KUKA KRL program: MyProgram_057().src

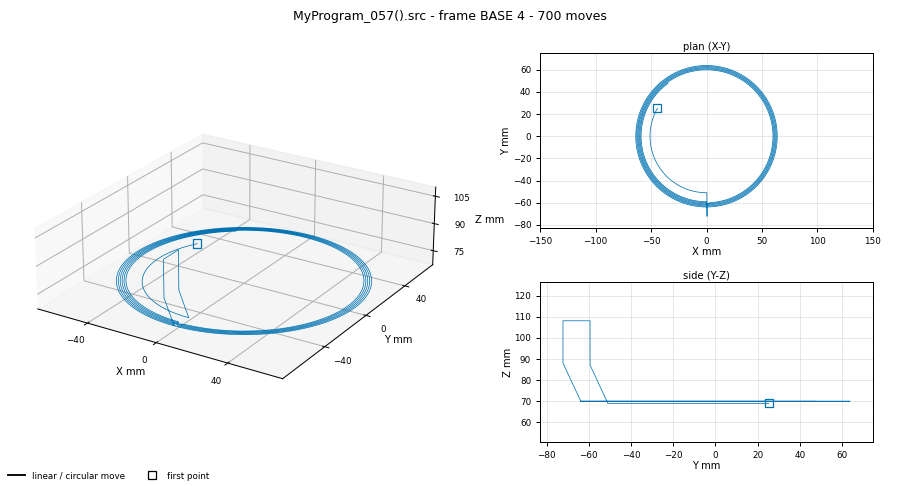
[picture p0: tool path of MyProgram_057().src in frame BASE 4, 700 of 700 moves have a stored position in this frame; points joined in program order, loops and branches not executed]
&ACCESS RVP
&REL 1
&PARAM TEMPLATE = C:\KRC\Roboter\Template\vorgabe
&PARAM EDITMASK = *
DEF MyProgram_057()
; ---- Setting reference (Base) ----
$BASE = BASE_DATA[4]

; --------------------------
; ---- Setting tool (TCP) ----
$TOOL = TOOL_DATA[3]
; --------------------------

$VEL.CP = VEL_APROX_PRINT
Startdeposition()
$VEL.CP = VEL_PRINT
LIN {X -44.2675,Y 25.2093,Z 69,A 144.3707,B 24.8543,C -2.785,E1 24.86,E2 299.1753} C_DIS
LIN {X -45.377,Y 23.1519,Z 69,A 147.0437,B 24.855,C -2.7781,E1 24.8565,E2 296.5045} C_DIS
LIN {X -46.4551,Y 20.9046,Z 69,A 149.9054,B 24.8558,C -2.7707,E1 24.8531,E2 293.6449} C_DIS
LIN {X -47.4216,Y 18.6083,Z 69,A 152.7265,B 24.8566,C -2.7626,E1 24.8502,E2 290.8275} C_DIS
LIN {X -48.2606,Y 16.3092,Z 69,A 155.5004,B 24.8575,C -2.7546,E1 24.8476,E2 288.057} C_DIS
LIN {X -49.0262,Y 13.8387,Z 69,A 158.4298,B 24.8584,C -2.7459,E1 24.8453,E2 285.1313} C_DIS
LIN {X -49.6447,Y 11.4229,Z 69,A 161.2158,B 24.8593,C -2.7369,E1 24.8435,E2 282.3505} C_DIS
LIN {X -50.1315,Y 9.0506,Z 69,A 163.9981,B 24.8601,C -2.7293,E1 24.842,E2 279.5701} C_DIS
LIN {X -50.5144,Y 6.5863,Z 69,A 166.8631,B 24.8609,C -2.7213,E1 24.8409,E2 276.707} C_DIS
LIN {X -50.7819,Y 4.0351,Z 69,A 169.7378,B 24.8619,C -2.7121,E1 24.8401,E2 273.8372} C_DIS
LIN {X -50.9193,Y 1.5178,Z 69,A 172.5271,B 24.8628,C -2.7025,E1 24.8398,E2 271.0541} C_DIS
LIN {X -50.9339,Y -0.9051,Z 69,A 175.3708,B 24.8635,C -2.6956,E1 24.8398,E2 268.2097} C_DIS
LIN {X -50.8236,Y -3.4697,Z 69,A 178.24,B 24.8645,C -2.6863,E1 24.8403,E2 265.3454} C_DIS
LIN {X -50.6012,Y -5.8824,Z 69,A -178.9757,B 24.8652,C -2.6787,E1 24.8411,E2 262.5626} C_DIS
LIN {X -50.2495,Y -8.3704,Z 69,A -176.13,B 24.8661,C -2.6703,E1 24.8423,E2 259.7201} C_DIS
LIN {X -49.7641,Y -10.891,Z 69,A -173.3005,B 24.8671,C -2.6607,E1 24.8439,E2 256.8968} C_DIS
LIN {X -49.1711,Y -13.3146,Z 69,A -170.4355,B 24.8678,C -2.6532,E1 24.8459,E2 254.0332} C_DIS
LIN {X -48.4775,Y -15.6528,Z 69,A -167.6344,B 24.8685,C -2.646,E1 24.8482,E2 251.2332} C_DIS
LIN {X -47.6271,Y -18.076,Z 69,A -164.8739,B 24.8696,C -2.6358,E1 24.8509,E2 248.4814} C_DIS
LIN {X -46.7092,Y -20.3305,Z 69,A -162.0822,B 24.8702,C -2.6289,E1 24.8539,E2 245.6908} C_DIS
LIN {X -45.6565,Y -22.5956,Z 69,A -159.1445,B 24.8708,C -2.6231,E1 24.8574,E2 242.751} C_DIS
LIN {X -44.4616,Y -24.8646,Z 69,A -156.2811,B 24.8716,C -2.6151,E1 24.8612,E2 239.8916} C_DIS
LIN {X -43.1923,Y -27.0093,Z 69,A -153.5018,B 24.8723,C -2.6075,E1 24.8653,E2 237.1162} C_DIS
LIN {X -41.8616,Y -29.0291,Z 69,A -150.6713,B 24.8728,C -2.6024,E1 24.8697,E2 234.2837} C_DIS
LIN {X -40.3456,Y -31.1016,Z 69,A -147.7568,B 24.8735,C -2.5959,E1 24.8746,E2 231.3707} C_DIS
LIN {X -38.6707,Y -33.1615,Z 69,A -144.8211,B 24.8742,C -2.5884,E1 24.8798,E2 228.4396} C_DIS
LIN {X -37.0149,Y -35,Z 69,A -142.0063,B 24.8748,C -2.5829,E1 24.8852,E2 225.6255} C_DIS
LIN {X -35.2304,Y -36.7958,Z 69,A -139.1593,B 24.8753,C -2.577,E1 24.8908,E2 222.7805} C_DIS
LIN {X -33.3921,Y -38.4716,Z 69,A -136.3039,B 24.8758,C -2.5726,E1 24.8968,E2 219.9244} C_DIS
LIN {X -31.3436,Y -40.1591,Z 69,A -133.3517,B 24.8763,C -2.5667,E1 24.9032,E2 216.9753} C_DIS
LIN {X -29.3388,Y -41.6462,Z 69,A -130.5429,B 24.8768,C -2.562,E1 24.9096,E2 214.1678} C_DIS
LIN {X -27.2507,Y -43.0415,Z 69,A -127.7018,B 24.8772,C -2.558,E1 24.9162,E2 211.3271} C_DIS
LIN {X -25.1158,Y -44.3212,Z 69,A -124.8909,B 24.8775,C -2.5543,E1 24.923,E2 208.5166} C_DIS
LIN {X -22.9218,Y -45.4946,Z 69,A -122.0757,B 24.8778,C -2.5511,E1 24.93,E2 205.7013} C_DIS
LIN {X -20.6449,Y -46.5721,Z 69,A -119.2428,B 24.8781,C -2.5479,E1 24.9372,E2 202.869} C_DIS
LIN {X -18.3398,Y -47.5271,Z 69,A -116.4302,B 24.8784,C -2.5453,E1 24.9445,E2 200.0564} C_DIS
LIN {X -15.9911,Y -48.3679,Z 69,A -113.6192,B 24.8786,C -2.5432,E1 24.9519,E2 197.2451} C_DIS
LIN {X -13.5856,Y -49.0979,Z 69,A -110.7884,B 24.8788,C -2.5413,E1 24.9595,E2 194.4141} C_DIS
LIN {X -11.1685,Y -49.7035,Z 69,A -107.9816,B 24.8788,C -2.54,E1 24.9671,E2 191.6066} C_DIS
LIN {X -8.7255,Y -50.19,Z 69,A -105.1777,B 24.879,C -2.5391,E1 24.9748,E2 188.802} C_DIS
LIN {X -6.264,Y -50.5561,Z 69,A -102.3662,B 24.879,C -2.5387,E1 24.9826,E2 185.9891} C_DIS
LIN {X -3.751,Y -50.8046,Z 69,A -99.5364,B 24.879,C -2.5384,E1 24.9905,E2 183.1587} C_DIS
LIN {X -1.2642,Y -50.9271,Z 69,A -96.7368,B 24.879,C -2.5387,E1 24.9983,E2 180.3579} C_DIS
LIN {X 0.3002,Y -50.939,Z 69,A -95.324,B 24.8796,C -2.5329,E1 25.0022,E2 178.9589} C_DIS
Enddeposition()
LIN {X 0.3252,Y -53.0519,Z 73.5315,A -95.3128,B 24.88,C -2.5282,E1 25.0022,E2 178.9589} C_DIS
LIN {X 0.4003,Y -59.3907,Z 87.1262,A -95.2837,B 24.8812,C -2.516,E1 25.0022,E2 178.9589} C_DIS
LIN {X 0.4003,Y -59.3907,Z 108.1262,A -95.6377,B 24.8666,C -2.6649,E1 25.0022,E2 178.9589} C_DIS
LIN {X 0.5021,Y -72.2249,Z 108.1262,A -95.1125,B 24.8869,C -2.4543,E1 25.0022,E2 178.9342} C_DIS
LIN {X 0.5021,Y -72.2249,Z 88.1262,A -94.7756,B 24.8997,C -2.3125,E1 25.0022,E2 178.9342} C_DIS
LIN {X 0.4243,Y -65.8861,Z 74.5315,A -94.8025,B 24.8987,C -2.3239,E1 25.0022,E2 178.9342} C_DIS
LIN {X 0.3983,Y -63.7731,Z 70,A -94.813,B 24.8983,C -2.3283,E1 25.0022,E2 178.9342} C_DIS
Startdeposition()
$VEL.CP = VEL_PRINT
LIN {X 3.1294,Y -63.7012,Z 70,A -92.0208,B 24.8975,C -2.3368,E1 25.0101,E2 176.1225} C_DIS
LIN {X 6.2513,Y -63.4709,Z 70,A -89.2116,B 24.8975,C -2.3382,E1 25.0179,E2 173.3116} C_DIS
LIN {X 9.3582,Y -63.0877,Z 70,A -86.4031,B 24.8973,C -2.3399,E1 25.0257,E2 170.5014} C_DIS
LIN {X 12.4425,Y -62.5525,Z 70,A -83.5957,B 24.8971,C -2.3421,E1 25.0334,E2 167.6921} C_DIS
LIN {X 15.4968,Y -61.8667,Z 70,A -80.7893,B 24.8969,C -2.3446,E1 25.0411,E2 164.8836} C_DIS
LIN {X 18.5138,Y -61.0318,Z 70,A -77.9838,B 24.8966,C -2.3475,E1 25.0486,E2 162.0759} C_DIS
LIN {X 21.4862,Y -60.0498,Z 70,A -75.1792,B 24.8963,C -2.3509,E1 25.056,E2 159.269} C_DIS
LIN {X 24.4068,Y -58.9232,Z 70,A -72.3755,B 24.896,C -2.3545,E1 25.0633,E2 156.4629} C_DIS
LIN {X 27.2686,Y -57.6546,Z 70,A -69.5725,B 24.8956,C -2.3586,E1 25.0704,E2 153.6573} C_DIS
LIN {X 30.0647,Y -56.2472,Z 70,A -66.7706,B 24.8952,C -2.363,E1 25.0773,E2 150.8527} C_DIS
LIN {X 32.7885,Y -54.7042,Z 70,A -63.9694,B 24.8948,C -2.3678,E1 25.0841,E2 148.0488} C_DIS
LIN {X 35.4332,Y -53.0295,Z 70,A -61.1691,B 24.8943,C -2.3729,E1 25.0907,E2 145.2456} C_DIS
LIN {X 37.9925,Y -51.227,Z 70,A -58.3694,B 24.8939,C -2.3783,E1 25.097,E2 142.443} C_DIS
LIN {X 40.4603,Y -49.3011,Z 70,A -55.5704,B 24.8933,C -2.384,E1 25.1031,E2 139.6409} C_DIS
LIN {X 42.8307,Y -47.2564,Z 70,A -52.7723,B 24.8928,C -2.39,E1 25.109,E2 136.8397} C_DIS
LIN {X 45.0979,Y -45.0979,Z 70,A -49.9747,B 24.8922,C -2.3963,E1 25.1146,E2 134.0389} C_DIS
LIN {X 47.2564,Y -42.8307,Z 70,A -47.1669,B 24.8916,C -2.4032,E1 25.1199,E2 131.2272} C_DIS
LIN {X 49.3011,Y -40.4603,Z 70,A -44.3816,B 24.891,C -2.4097,E1 25.1249,E2 128.4392} C_DIS
LIN {X 51.227,Y -37.9925,Z 70,A -41.5858,B 24.8904,C -2.4168,E1 25.1296,E2 125.64} C_DIS
LIN {X 53.0295,Y -35.4332,Z 70,A -38.7905,B 24.8897,C -2.424,E1 25.1341,E2 122.8413} C_DIS
LIN {X 54.7042,Y -32.7885,Z 70,A -35.9957,B 24.889,C -2.4315,E1 25.1382,E2 120.0431} C_DIS
LIN {X 56.2472,Y -30.0647,Z 70,A -33.2013,B 24.8883,C -2.4391,E1 25.1419,E2 117.2453} C_DIS
LIN {X 57.6546,Y -27.2686,Z 70,A -30.4073,B 24.8876,C -2.4469,E1 25.1454,E2 114.4478} C_DIS
LIN {X 58.9232,Y -24.4068,Z 70,A -27.6138,B 24.8869,C -2.4548,E1 25.1484,E2 111.6509} C_DIS
LIN {X 60.0498,Y -21.4862,Z 70,A -24.8204,B 24.8862,C -2.4629,E1 25.1511,E2 108.8541} C_DIS
LIN {X 61.0318,Y -18.5138,Z 70,A -22.0273,B 24.8854,C -2.4711,E1 25.1535,E2 106.0575} C_DIS
LIN {X 61.8667,Y -15.4968,Z 70,A -19.2344,B 24.8846,C -2.4793,E1 25.1555,E2 103.2611} C_DIS
LIN {X 62.5525,Y -12.4425,Z 70,A -16.4416,B 24.8838,C -2.4876,E1 25.1571,E2 100.465} C_DIS
LIN {X 63.0877,Y -9.3582,Z 70,A -13.6491,B 24.8831,C -2.496,E1 25.1583,E2 97.6691} C_DIS
LIN {X 63.4709,Y -6.2513,Z 70,A -10.8566,B 24.8823,C -2.5044,E1 25.1592,E2 94.8733} C_DIS
LIN {X 63.7012,Y -3.1294,Z 70,A -8.0639,B 24.8815,C -2.5128,E1 25.1597,E2 92.0774} C_DIS
LIN {X 63.7798,Y 0.0603,Z 70,A -5.1773,B 24.8806,C -2.5224,E1 25.1597,E2 89.1853} C_DIS
LIN {X 63.7012,Y 3.1294,Z 70,A -2.4788,B 24.8799,C -2.5295,E1 25.1595,E2 86.4859} C_DIS
LIN {X 63.4709,Y 6.2513,Z 70,A 0.314,B 24.8791,C -2.5378,E1 25.1588,E2 83.69} C_DIS
LIN {X 63.0877,Y 9.3582,Z 70,A 3.107,B 24.8783,C -2.5461,E1 25.1578,E2 80.8941} C_DIS
LIN {X 62.5525,Y 12.4425,Z 70,A 5.9002,B 24.8775,C -2.5542,E1 25.1563,E2 78.098} C_DIS
LIN {X 61.8667,Y 15.4968,Z 70,A 8.6935,B 24.8768,C -2.5622,E1 25.1545,E2 75.3018} C_DIS
LIN {X 61.0318,Y 18.5138,Z 70,A 11.4872,B 24.876,C -2.5701,E1 25.1523,E2 72.5055} C_DIS
LIN {X 60.0498,Y 21.4862,Z 70,A 14.2814,B 24.8752,C -2.5779,E1 25.1498,E2 69.7087} C_DIS
LIN {X 58.9232,Y 24.4068,Z 70,A 17.0758,B 24.8745,C -2.5855,E1 25.1469,E2 66.9118} C_DIS
LIN {X 57.6546,Y 27.2686,Z 70,A 19.8708,B 24.8738,C -2.5929,E1 25.1436,E2 64.1144} C_DIS
LIN {X 56.2472,Y 30.0647,Z 70,A 22.6661,B 24.8731,C -2.6,E1 25.14,E2 61.3169} C_DIS
LIN {X 54.7042,Y 32.7885,Z 70,A 25.4621,B 24.8724,C -2.607,E1 25.1361,E2 58.5189} C_DIS
LIN {X 53.0295,Y 35.4332,Z 70,A 28.2585,B 24.8717,C -2.6138,E1 25.1318,E2 55.7205} C_DIS
LIN {X 51.227,Y 37.9925,Z 70,A 31.0556,B 24.8711,C -2.6202,E1 25.1273,E2 52.9216} C_DIS
LIN {X 49.3011,Y 40.4603,Z 70,A 33.8533,B 24.8705,C -2.6265,E1 25.1224,E2 50.1222} C_DIS
LIN {X 47.2564,Y 42.8307,Z 70,A 36.6518,B 24.8699,C -2.6324,E1 25.1172,E2 47.3223} C_DIS
LIN {X 45.0979,Y 45.0979,Z 70,A 39.4508,B 24.8693,C -2.638,E1 25.1117,E2 44.5219} C_DIS
LIN {X 42.8307,Y 47.2564,Z 70,A 42.2506,B 24.8688,C -2.6433,E1 25.106,E2 41.7209} C_DIS
LIN {X 40.4603,Y 49.3011,Z 70,A 45.0513,B 24.8683,C -2.6483,E1 25.1,E2 38.9192} C_DIS
LIN {X 37.9925,Y 51.227,Z 70,A 47.8528,B 24.8678,C -2.653,E1 25.0938,E2 36.1168} C_DIS
LIN {X 35.4332,Y 53.0295,Z 70,A 50.6549,B 24.8674,C -2.6573,E1 25.0873,E2 33.314} C_DIS
LIN {X 32.7885,Y 54.7042,Z 70,A 53.458,B 24.867,C -2.6613,E1 25.0807,E2 30.5104} C_DIS
LIN {X 30.0647,Y 56.2472,Z 70,A 56.262,B 24.8666,C -2.6649,E1 25.0738,E2 27.706} C_DIS
LIN {X 27.2686,Y 57.6546,Z 70,A 59.0668,B 24.8663,C -2.6681,E1 25.0668,E2 24.901} C_DIS
LIN {X 24.4068,Y 58.9232,Z 70,A 61.8725,B 24.866,C -2.6709,E1 25.0596,E2 22.0953} C_DIS
LIN {X 21.4862,Y 60.0498,Z 70,A 64.6793,B 24.8658,C -2.6734,E1 25.0522,E2 19.2886} C_DIS
LIN {X 18.5138,Y 61.0318,Z 70,A 67.4869,B 24.8656,C -2.6754,E1 25.0447,E2 16.4813} C_DIS
LIN {X 15.4968,Y 61.8667,Z 70,A 70.2955,B 24.8654,C -2.6771,E1 25.0371,E2 13.6731} C_DIS
LIN {X 12.4425,Y 62.5525,Z 70,A 73.1051,B 24.8653,C -2.6783,E1 25.0295,E2 10.8642} C_DIS
LIN {X 9.3582,Y 63.0877,Z 70,A 75.9156,B 24.8653,C -2.6791,E1 25.0217,E2 8.0545} C_DIS
LIN {X 6.2513,Y 63.4709,Z 70,A 78.727,B 24.8652,C -2.6795,E1 25.0139,E2 5.2441} C_DIS
LIN {X 3.1294,Y 63.7012,Z 70,A 81.5396,B 24.8652,C -2.6795,E1 25.0061,E2 2.4326} C_DIS
LIN {X 0,Y 63.778,Z 70,A 84.3531,B 24.8652,C -2.6791,E1 24.9982,E2 -0.3796} C_DIS
LIN {X -3.1294,Y 63.7012,Z 70,A 87.1675,B 24.8652,C -2.6783,E1 24.9904,E2 -3.1926} C_DIS
LIN {X -6.2513,Y 63.4709,Z 70,A 89.9829,B 24.8654,C -2.6771,E1 24.9826,E2 -6.0064} C_DIS
LIN {X -9.3582,Y 63.0877,Z 70,A 92.7995,B 24.8656,C -2.6754,E1 24.9748,E2 -8.8211} C_DIS
LIN {X -12.4425,Y 62.5525,Z 70,A 95.6169,B 24.8658,C -2.6734,E1 24.967,E2 -11.6366} C_DIS
LIN {X -15.4968,Y 61.8667,Z 70,A 98.4352,B 24.866,C -2.6709,E1 24.9594,E2 -14.4529} C_DIS
LIN {X -18.5138,Y 61.0318,Z 70,A 101.2544,B 24.8663,C -2.6681,E1 24.9518,E2 -17.27} C_DIS
LIN {X -21.4861,Y 60.0497,Z 70,A 104.0712,B 24.8667,C -2.6647,E1 24.9444,E2 -20.0842} C_DIS
LIN {X -24.4068,Y 58.9232,Z 70,A 106.8957,B 24.867,C -2.6612,E1 24.9371,E2 -22.9065} C_DIS
LIN {X -27.2686,Y 57.6546,Z 70,A 109.7178,B 24.8674,C -2.6572,E1 24.9299,E2 -25.7261} C_DIS
LIN {X -30.0647,Y 56.2472,Z 70,A 112.5406,B 24.8679,C -2.6528,E1 24.9229,E2 -28.5462} C_DIS
LIN {X -32.7885,Y 54.7042,Z 70,A 115.3643,B 24.8683,C -2.6481,E1 24.9161,E2 -31.3671} C_DIS
LIN {X -35.4332,Y 53.0295,Z 70,A 118.1889,B 24.8688,C -2.6431,E1 24.9095,E2 -34.1888} C_DIS
LIN {X -37.9925,Y 51.227,Z 70,A 121.0141,B 24.8694,C -2.6377,E1 24.9032,E2 -37.0111} C_DIS
LIN {X -40.4603,Y 49.3011,Z 70,A 123.8402,B 24.8699,C -2.632,E1 24.897,E2 -39.8341} C_DIS
LIN {X -42.8307,Y 47.2564,Z 70,A 126.6669,B 24.8705,C -2.626,E1 24.8911,E2 -42.6577} C_DIS
LIN {X -45.0979,Y 45.0979,Z 70,A 129.4944,B 24.8711,C -2.6197,E1 24.8855,E2 -45.482} C_DIS
LIN {X -47.2564,Y 42.8307,Z 70,A 132.3225,B 24.8718,C -2.6131,E1 24.8801,E2 -48.3068} C_DIS
LIN {X -49.3011,Y 40.4603,Z 70,A 135.1512,B 24.8725,C -2.6063,E1 24.875,E2 -51.1322} C_DIS
LIN {X -51.227,Y 37.9925,Z 70,A 137.9805,B 24.8732,C -2.5992,E1 24.8702,E2 -53.9582} C_DIS
LIN {X -53.0295,Y 35.4332,Z 70,A 140.8102,B 24.8739,C -2.592,E1 24.8658,E2 -56.7845} C_DIS
LIN {X -54.7042,Y 32.7885,Z 70,A 143.6407,B 24.8746,C -2.5845,E1 24.8616,E2 -59.6115} C_DIS
LIN {X -56.2472,Y 30.0647,Z 70,A 146.4715,B 24.8753,C -2.5768,E1 24.8578,E2 -62.4389} C_DIS
LIN {X -57.6546,Y 27.2686,Z 70,A 149.3027,B 24.8761,C -2.5689,E1 24.8544,E2 -65.2666} C_DIS
LIN {X -58.9232,Y 24.4068,Z 70,A 152.1342,B 24.8769,C -2.5609,E1 24.8513,E2 -68.0946} C_DIS
LIN {X -60.0498,Y 21.4862,Z 70,A 154.966,B 24.8777,C -2.5528,E1 24.8485,E2 -70.923} C_DIS
LIN {X -61.0318,Y 18.5138,Z 70,A 157.7981,B 24.8785,C -2.5445,E1 24.8461,E2 -73.7516} C_DIS
LIN {X -61.8667,Y 15.4968,Z 70,A 160.6305,B 24.8793,C -2.5362,E1 24.8441,E2 -76.5805} C_DIS
LIN {X -62.5525,Y 12.4425,Z 70,A 163.463,B 24.8801,C -2.5278,E1 24.8425,E2 -79.4096} C_DIS
LIN {X -63.0877,Y 9.3582,Z 70,A 166.2956,B 24.8809,C -2.5193,E1 24.8412,E2 -82.2388} C_DIS
LIN {X -63.4709,Y 6.2513,Z 70,A 169.1282,B 24.8817,C -2.5108,E1 24.8404,E2 -85.0681} C_DIS
LIN {X -63.7012,Y 3.1294,Z 70,A 171.961,B 24.8825,C -2.5023,E1 24.8399,E2 -87.8976} C_DIS
LIN {X -63.7798,Y -0.0603,Z 70,A 174.8891,B 24.8832,C -2.4944,E1 24.8398,E2 -90.8245} C_DIS
LIN {X -63.7012,Y -3.1294,Z 70,A 177.6262,B 24.8841,C -2.4854,E1 24.8401,E2 -93.5565} C_DIS
LIN {X -63.4709,Y -6.2513,Z 70,A -179.5413,B 24.8848,C -2.477,E1 24.8408,E2 -96.3858} C_DIS
LIN {X -63.0877,Y -9.3582,Z 70,A -176.709,B 24.8856,C -2.4686,E1 24.8418,E2 -99.2152} C_DIS
LIN {X -62.5525,Y -12.4425,Z 70,A -173.8769,B 24.8864,C -2.4604,E1 24.8433,E2 -102.0444} C_DIS
LIN {X -61.8667,Y -15.4968,Z 70,A -171.0451,B 24.8871,C -2.4523,E1 24.8451,E2 -104.8734} C_DIS
LIN {X -61.0318,Y -18.5138,Z 70,A -168.2137,B 24.8879,C -2.4443,E1 24.8473,E2 -107.7021} C_DIS
LIN {X -60.0498,Y -21.4862,Z 70,A -165.3826,B 24.8886,C -2.4365,E1 24.8499,E2 -110.5305} C_DIS
LIN {X -58.9232,Y -24.4068,Z 70,A -162.5519,B 24.8893,C -2.4288,E1 24.8528,E2 -113.3588} C_DIS
LIN {X -57.6546,Y -27.2686,Z 70,A -159.7216,B 24.89,C -2.4213,E1 24.8561,E2 -116.1868} C_DIS
LIN {X -56.2472,Y -30.0647,Z 70,A -156.8919,B 24.8906,C -2.4141,E1 24.8597,E2 -119.0142} C_DIS
LIN {X -54.7042,Y -32.7885,Z 70,A -154.0627,B 24.8913,C -2.4071,E1 24.8637,E2 -121.8413} C_DIS
LIN {X -53.0295,Y -35.4332,Z 70,A -151.2342,B 24.8919,C -2.4003,E1 24.868,E2 -124.6679} C_DIS
LIN {X -51.227,Y -37.9925,Z 70,A -148.4062,B 24.8925,C -2.3938,E1 24.8727,E2 -127.4941} C_DIS
LIN {X -49.3011,Y -40.4603,Z 70,A -145.5788,B 24.893,C -2.3875,E1 24.8776,E2 -130.3199} C_DIS
LIN {X -47.2564,Y -42.8307,Z 70,A -142.7522,B 24.8936,C -2.3816,E1 24.8828,E2 -133.1449} C_DIS
LIN {X -45.0979,Y -45.0979,Z 70,A -139.9263,B 24.8941,C -2.3759,E1 24.8883,E2 -135.9695} C_DIS
LIN {X -42.8307,Y -47.2564,Z 70,A -137.1011,B 24.8945,C -2.3706,E1 24.8941,E2 -138.7935} C_DIS
LIN {X -40.4603,Y -49.3011,Z 70,A -134.2769,B 24.895,C -2.3656,E1 24.9001,E2 -141.6167} C_DIS
LIN {X -37.9925,Y -51.227,Z 70,A -131.4533,B 24.8954,C -2.361,E1 24.9064,E2 -144.4394} C_DIS
LIN {X -35.4332,Y -53.0295,Z 70,A -128.6306,B 24.8958,C -2.3567,E1 24.9129,E2 -147.2614} C_DIS
LIN {X -32.7885,Y -54.7042,Z 70,A -125.8088,B 24.8961,C -2.3528,E1 24.9196,E2 -150.0827} C_DIS
LIN {X -30.0647,Y -56.2472,Z 70,A -122.9879,B 24.8964,C -2.3493,E1 24.9265,E2 -152.9033} C_DIS
LIN {X -27.2686,Y -57.6546,Z 70,A -120.1678,B 24.8967,C -2.3461,E1 24.9336,E2 -155.7231} C_DIS
LIN {X -24.4068,Y -58.9232,Z 70,A -117.3489,B 24.897,C -2.3433,E1 24.9408,E2 -158.542} C_DIS
LIN {X -21.4862,Y -60.0498,Z 70,A -114.5307,B 24.8972,C -2.341,E1 24.9482,E2 -161.3603} C_DIS
LIN {X -18.5138,Y -61.0318,Z 70,A -111.7135,B 24.8973,C -2.339,E1 24.9557,E2 -164.1779} C_DIS
LIN {X -15.4968,Y -61.8667,Z 70,A -108.8973,B 24.8975,C -2.3374,E1 24.9633,E2 -166.9946} C_DIS
LIN {X -12.4425,Y -62.5525,Z 70,A -106.082,B 24.8975,C -2.3363,E1 24.971,E2 -169.8105} C_DIS
LIN {X -9.3582,Y -63.0877,Z 70,A -103.2679,B 24.8976,C -2.3356,E1 24.9788,E2 -172.6255} C_DIS
LIN {X -6.2513,Y -63.4709,Z 70,A -100.4547,B 24.8976,C -2.3353,E1 24.9866,E2 -175.4397} C_DIS
LIN {X -3.1294,Y -63.7012,Z 70,A -97.6423,B 24.8976,C -2.3353,E1 24.9944,E2 -178.2532} C_DIS
LIN {X 0,Y -63.778,Z 70,A -94.8311,B 24.8976,C -2.3359,E1 25.0023,E2 -181.0657} C_DIS
LIN {X 0,Y -63.778,Z 70,A -94.8311,B 24.8976,C -2.3359,E1 25.0023,E2 -181.0657} C_DIS
Enddeposition()
LIN {X 0.3983,Y -62.8225,Z 70,A -95.5183,B 24.8982,C -2.3289,E1 25.0003,E2 -180.3619} C_DIS
Startdeposition()
$VEL.CP = VEL_PRINT
LIN {X -2.2693,Y -62.7853,Z 70,A -98.2915,B 24.8989,C -2.321,E1 24.9925,E2 -177.5696} C_DIS
LIN {X -5.4728,Y -62.5872,Z 70,A -101.2578,B 24.899,C -2.3201,E1 24.9842,E2 -174.6002} C_DIS
LIN {X -8.5647,Y -62.2395,Z 70,A -104.3097,B 24.8994,C -2.316,E1 24.9758,E2 -171.5363} C_DIS
LIN {X -11.1905,Y -61.8208,Z 70,A -106.4634,B 24.8988,C -2.3226,E1 24.9699,E2 -169.3961} C_DIS
LIN {X -14.0107,Y -61.2434,Z 70,A -109.0327,B 24.8986,C -2.3249,E1 24.9629,E2 -166.8293} C_DIS
LIN {X -16.9205,Y -60.5043,Z 70,A -111.8232,B 24.8986,C -2.3254,E1 24.9553,E2 -164.0358} C_DIS
LIN {X -20.0863,Y -59.5279,Z 70,A -114.6327,B 24.8979,C -2.3322,E1 24.9479,E2 -161.2372} C_DIS
LIN {X -23.3407,Y -58.3278,Z 70,A -118.0164,B 24.8981,C -2.3304,E1 24.939,E2 -157.8423} C_DIS
LIN {X -26.2064,Y -57.0978,Z 70,A -121.1327,B 24.8983,C -2.3279,E1 24.931,E2 -154.7124} C_DIS
LIN {X -29.5531,Y -55.4414,Z 70,A -124.038,B 24.8971,C -2.3423,E1 24.9239,E2 -151.8337} C_DIS
LIN {X -31.4318,Y -54.3976,Z 70,A -126.1261,B 24.8971,C -2.3423,E1 24.9188,E2 -149.7396} C_DIS
LIN {X -34.3527,Y -52.6023,Z 70,A -129.1071,B 24.8964,C -2.35,E1 24.9118,E2 -146.7673} C_DIS
LIN {X -36.4245,Y -51.1888,Z 70,A -131.6531,B 24.8965,C -2.3485,E1 24.9059,E2 -144.209} C_DIS
LIN {X -38.5528,Y -49.6062,Z 70,A -134.0836,B 24.8962,C -2.3524,E1 24.9005,E2 -141.7792} C_DIS
LIN {X -40.3962,Y -48.1173,Z 70,A -136.0864,B 24.8955,C -2.3595,E1 24.8962,E2 -139.7857} C_DIS
LIN {X -42.1519,Y -46.5871,Z 70,A -138.481,B 24.8956,C -2.3583,E1 24.8912,E2 -137.3786} C_DIS
LIN {X -44.322,Y -44.527,Z 70,A -141.125,B 24.895,C -2.3655,E1 24.8859,E2 -134.7409} C_DIS
LIN {X -46.14,Y -42.6397,Z 70,A -144.1002,B 24.8955,C -2.3593,E1 24.8802,E2 -131.7379} C_DIS
LIN {X -49.6526,Y -38.4926,Z 70,A -148.364,B 24.8933,C -2.3841,E1 24.8727,E2 -127.5134} C_DIS
LIN {X -50.7082,Y -37.0906,Z 70,A -150.0283,B 24.8931,C -2.3867,E1 24.8699,E2 -125.8473} C_DIS
LIN {X -52.1818,Y -34.9882,Z 70,A -152.4574,B 24.8927,C -2.3908,E1 24.8661,E2 -123.416} C_DIS
LIN {X -53.5978,Y -32.7771,Z 70,A -154.9256,B 24.8923,C -2.3956,E1 24.8624,E2 -120.9465} C_DIS
LIN {X -55.2237,Y -29.9561,Z 70,A -157.837,B 24.8915,C -2.4045,E1 24.8585,E2 -118.0413} C_DIS
LIN {X -56.462,Y -27.554,Z 70,A -160.3439,B 24.891,C -2.4104,E1 24.8553,E2 -115.535} C_DIS
LIN {X -57.7476,Y -24.7464,Z 70,A -163.0379,B 24.89,C -2.4206,E1 24.8523,E2 -112.8505} C_DIS
LIN {X -58.6136,Y -22.6191,Z 70,A -165.4132,B 24.89,C -2.4213,E1 24.8498,E2 -110.4636} C_DIS
LIN {X -59.6225,Y -19.8056,Z 70,A -168.0186,B 24.889,C -2.4315,E1 24.8475,E2 -107.8678} C_DIS
LIN {X -60.4741,Y -17.0271,Z 70,A -170.6842,B 24.8883,C -2.4391,E1 24.8453,E2 -105.2049} C_DIS
LIN {X -61.1611,Y -14.3666,Z 70,A -173.1767,B 24.8876,C -2.4469,E1 24.8437,E2 -102.7164} C_DIS
LIN {X -61.7294,Y -11.6857,Z 70,A -175.7899,B 24.8871,C -2.4524,E1 24.8422,E2 -100.101} C_DIS
LIN {X -62.2334,Y -8.6073,Z 70,A -179.4438,B 24.8877,C -2.4464,E1 24.8408,E2 -96.411} C_DIS
LIN {X -62.6034,Y -5.2846,Z 70,A 178.699,B 24.8848,C -2.4778,E1 24.8403,E2 -94.6175} C_DIS
LIN {X -62.8256,Y 0.3633,Z 70,A 173.1574,B 24.8839,C -2.4869,E1 24.8398,E2 -89.0642} C_DIS
LIN {X -62.7462,Y 3.167,Z 70,A 170.5757,B 24.8832,C -2.4945,E1 24.8401,E2 -86.4853} C_DIS
LIN {X -62.5441,Y 5.9407,Z 70,A 168.0003,B 24.8825,C -2.5018,E1 24.8407,E2 -83.9119} C_DIS
LIN {X -62.0366,Y 9.93,Z 70,A 164.594,B 24.881,C -2.5182,E1 24.842,E2 -80.5244} C_DIS
LIN {X -61.7007,Y 11.8342,Z 70,A 162.2601,B 24.8814,C -2.5133,E1 24.8432,E2 -78.1649} C_DIS
LIN {X -60.7801,Y 15.9024,Z 70,A 158.6031,B 24.8801,C -2.5278,E1 24.8455,E2 -74.5212} C_DIS
LIN {X -59.875,Y 19.0295,Z 70,A 155.7387,B 24.879,C -2.5388,E1 24.8479,E2 -71.6667} C_DIS
LIN {X -59.0404,Y 21.4771,Z 70,A 153.3003,B 24.8785,C -2.5446,E1 24.8501,E2 -69.2282} C_DIS
LIN {X -58.2776,Y 23.4692,Z 70,A 151.4582,B 24.8777,C -2.5523,E1 24.852,E2 -67.3943} C_DIS
LIN {X -56.895,Y 26.646,Z 70,A 148.4665,B 24.8765,C -2.5648,E1 24.8554,E2 -64.416} C_DIS
LIN {X -55.8676,Y 28.7379,Z 70,A 146.0338,B 24.8765,C -2.5653,E1 24.8584,E2 -61.9713} C_DIS
LIN {X -54.5016,Y 31.2507,Z 70,A 143.4218,B 24.8757,C -2.5726,E1 24.862,E2 -59.3632} C_DIS
LIN {X -52.9628,Y 33.7935,Z 70,A 140.7356,B 24.875,C -2.5806,E1 24.8659,E2 -56.6824} C_DIS
LIN {X -50.8792,Y 36.8564,Z 70,A 137.2585,B 24.8743,C -2.5879,E1 24.8715,E2 -53.2056} C_DIS
LIN {X -49.0194,Y 39.2968,Z 70,A 134.423,B 24.8736,C -2.5945,E1 24.8764,E2 -50.3725} C_DIS
LIN {X -47.0287,Y 41.6586,Z 70,A 131.6926,B 24.8728,C -2.6032,E1 24.8813,E2 -47.6505} C_DIS
LIN {X -45.3149,Y 43.5155,Z 70,A 129.3676,B 24.8722,C -2.6085,E1 24.8858,E2 -45.3278} C_DIS
LIN {X -43.3919,Y 45.4341,Z 70,A 126.7843,B 24.8719,C -2.6122,E1 24.8909,E2 -42.7428} C_DIS
LIN {X -41.0723,Y 47.5417,Z 70,A 124.0037,B 24.8711,C -2.6201,E1 24.8967,E2 -39.9699} C_DIS
LIN {X -39.1425,Y 49.1422,Z 70,A 121.7406,B 24.8706,C -2.6255,E1 24.9016,E2 -37.7111} C_DIS
LIN {X -37.1141,Y 50.6909,Z 70,A 119.4238,B 24.8701,C -2.6305,E1 24.9068,E2 -35.3979} C_DIS
LIN {X -34.9108,Y 52.2339,Z 70,A 116.8616,B 24.8698,C -2.6331,E1 24.9127,E2 -32.8333} C_DIS
LIN {X -32.5963,Y 53.7076,Z 70,A 114.3767,B 24.8693,C -2.638,E1 24.9186,E2 -30.3523} C_DIS
LIN {X -30.1851,Y 55.0995,Z 70,A 111.8277,B 24.8689,C -2.6422,E1 24.9248,E2 -27.8058} C_DIS
LIN {X -27.6184,Y 56.4301,Z 70,A 109.1007,B 24.8687,C -2.6446,E1 24.9316,E2 -25.0773} C_DIS
LIN {X -24.2492,Y 57.9572,Z 70,A 105.9168,B 24.8678,C -2.6533,E1 24.9397,E2 -21.9065} C_DIS
LIN {X -20.8668,Y 59.2588,Z 70,A 102.1311,B 24.8683,C -2.6479,E1 24.9496,E2 -18.1001} C_DIS
LIN {X -17.4964,Y 60.3411,Z 70,A 98.6384,B 24.8685,C -2.646,E1 24.959,E2 -14.5972} C_DIS
LIN {X -12.2949,Y 61.6116,Z 70,A 94.2773,B 24.867,C -2.661,E1 24.9708,E2 -10.2662} C_DIS
LIN {X -9.2382,Y 62.1435,Z 70,A 91.472,B 24.8668,C -2.6635,E1 24.9785,E2 -7.4642} C_DIS
LIN {X -5.0007,Y 62.6261,Z 70,A 87.6286,B 24.8665,C -2.6665,E1 24.9892,E2 -3.6258} C_DIS
LIN {X -2.7616,Y 62.7647,Z 70,A 85.5241,B 24.8665,C -2.666,E1 24.9951,E2 -1.5195} C_DIS
LIN {X 0.2278,Y 62.8252,Z 70,A 82.7828,B 24.8665,C -2.6663,E1 25.0027,E2 1.2211} C_DIS
LIN {X 3.3874,Y 62.7341,Z 70,A 79.9827,B 24.8663,C -2.6683,E1 25.0105,E2 4.0158} C_DIS
LIN {X 6.1367,Y 62.526,Z 70,A 77.071,B 24.8672,C -2.6595,E1 25.0187,E2 6.9467} C_DIS
LIN {X 9.1813,Y 62.1519,Z 70,A 74.6103,B 24.8665,C -2.6661,E1 25.0254,E2 9.3896} C_DIS
LIN {X 11.9643,Y 61.6757,Z 70,A 72.0551,B 24.8665,C -2.6656,E1 25.0324,E2 11.9432} C_DIS
LIN {X 14.9586,Y 61.0187,Z 70,A 69.111,B 24.867,C -2.6609,E1 25.0405,E2 14.8944} C_DIS
LIN {X 18.3199,Y 60.0958,Z 70,A 65.7822,B 24.8676,C -2.6553,E1 25.0494,E2 18.2306} C_DIS
LIN {X 21.9214,Y 58.8779,Z 70,A 62.5253,B 24.8674,C -2.657,E1 25.0579,E2 21.4769} C_DIS
LIN {X 25.4804,Y 57.4274,Z 70,A 59.129,B 24.8676,C -2.6558,E1 25.0667,E2 24.8681} C_DIS
LIN {X 27.5881,Y 56.4451,Z 70,A 56.9366,B 24.868,C -2.6516,E1 25.0722,E2 27.0647} C_DIS
LIN {X 31.3179,Y 54.463,Z 70,A 53.1174,B 24.8684,C -2.6472,E1 25.0816,E2 30.8832} C_DIS
LIN {X 33.9718,Y 52.8483,Z 70,A 50.2764,B 24.8689,C -2.6428,E1 25.0883,E2 33.7256} C_DIS
LIN {X 37.6365,Y 50.3043,Z 70,A 46.5852,B 24.8687,C -2.6448,E1 25.0967,E2 37.3993} C_DIS
LIN {X 39.3276,Y 48.9945,Z 70,A 44.3866,B 24.8696,C -2.6355,E1 25.1015,E2 39.6118} C_DIS
LIN {X 41.4657,Y 47.1981,Z 70,A 41.7517,B 24.8703,C -2.6286,E1 25.1071,E2 42.2528} C_DIS
LIN {X 43.2288,Y 45.5891,Z 70,A 39.6506,B 24.8705,C -2.626,E1 25.1114,E2 44.3514} C_DIS
LIN {X 45.219,Y 43.615,Z 70,A 37.1388,B 24.8709,C -2.6217,E1 25.1163,E2 46.8627} C_DIS
LIN {X 47.9633,Y 40.5783,Z 70,A 33.607,B 24.8713,C -2.6182,E1 25.1228,E2 50.3871} C_DIS
LIN {X 49.468,Y 38.7302,Z 70,A 31.2323,B 24.8723,C -2.6082,E1 25.127,E2 52.7741} C_DIS
LIN {X 51.135,Y 36.5,Z 70,A 28.5353,B 24.8733,C -2.5983,E1 25.1315,E2 55.4817} C_DIS
LIN {X 52.7405,Y 34.1399,Z 70,A 26.1154,B 24.8735,C -2.5961,E1 25.1352,E2 57.8947} C_DIS
LIN {X 54.2727,Y 31.6486,Z 70,A 22.6566,B 24.876,C -2.57,E1 25.1401,E2 61.3975} C_DIS
LIN {X 55.843,Y 28.786,Z 70,A 20.4654,B 24.8749,C -2.581,E1 25.1429,E2 63.5509} C_DIS
LIN {X 57.1813,Y 26.0267,Z 70,A 17.7654,B 24.8755,C -2.5757,E1 25.1462,E2 66.2492} C_DIS
LIN {X 59.0448,Y 21.4649,Z 70,A 13.6042,B 24.8759,C -2.571,E1 25.1505,E2 70.3983} C_DIS
LIN {X 59.7241,Y 19.4957,Z 70,A 11.3589,B 24.8773,C -2.5569,E1 25.1525,E2 72.6643} C_DIS
LIN {X 60.6416,Y 16.4204,Z 70,A 8.0961,B 24.8789,C -2.5399,E1 25.155,E2 75.9486} C_DIS
LIN {X 61.5996,Y 12.3532,Z 70,A 4.735,B 24.8789,C -2.5394,E1 25.157,E2 79.2913} C_DIS
LIN {X 62.0764,Y 9.6723,Z 70,A 2.162,B 24.8799,C -2.5296,E1 25.1582,E2 81.8725} C_DIS
LIN {X 62.5407,Y 5.9772,Z 70,A -1.0644,B 24.8805,C -2.5232,E1 25.1592,E2 85.0948} C_DIS
LIN {X 62.7517,Y 3.0621,Z 70,A -3.8919,B 24.8817,C -2.5108,E1 25.1597,E2 87.9348} C_DIS
LIN {X 62.8281,Y -0.093,Z 70,A -6.7148,B 24.8824,C -2.5031,E1 25.1597,E2 90.7592} C_DIS
LIN {X 62.7546,Y -2.9969,Z 70,A -9.2789,B 24.883,C -2.4968,E1 25.1595,E2 93.3228} C_DIS
LIN {X 62.5648,Y -5.7168,Z 70,A -11.6597,B 24.8835,C -2.4916,E1 25.159,E2 95.7019} C_DIS
LIN {X 62.3693,Y -7.5608,Z 70,A -13.4474,B 24.8842,C -2.4838,E1 25.1584,E2 97.4974} C_DIS
LIN {X 61.9743,Y -10.3063,Z 70,A -15.9192,B 24.8848,C -2.4773,E1 25.1573,E2 99.9701} C_DIS
LIN {X 61.4575,Y -13.0431,Z 70,A -18.7755,B 24.8863,C -2.4614,E1 25.1558,E2 102.8473} C_DIS
LIN {X 60.7372,Y -16.0663,Z 70,A -21.3599,B 24.8865,C -2.4588,E1 25.154,E2 105.4229} C_DIS
LIN {X 59.5419,Y -20.0447,Z 70,A -24.4801,B 24.8861,C -2.4638,E1 25.1515,E2 108.5134} C_DIS
LIN {X 58.8794,Y -21.9174,Z 70,A -26.9257,B 24.888,C -2.4424,E1 25.1491,E2 110.9959} C_DIS
LIN {X 57.7355,Y -24.7744,Z 70,A -29.6649,B 24.8887,C -2.4357,E1 25.1462,E2 113.736} C_DIS
LIN {X 55.9204,Y -28.6346,Z 70,A -33.3085,B 24.8891,C -2.4304,E1 25.1418,E2 117.3725} C_DIS
LIN {X 55.1226,Y -30.1426,Z 70,A -35.0162,B 24.8899,C -2.4221,E1 25.1395,E2 119.0909} C_DIS
LIN {X 53.8189,Y -32.4133,Z 70,A -37.3721,B 24.8904,C -2.4161,E1 25.1361,E2 121.4488} C_DIS
LIN {X 52.4431,Y -34.5941,Z 70,A -39.7243,B 24.891,C -2.4096,E1 25.1326,E2 123.8047} C_DIS
LIN {X 50.8163,Y -36.9429,Z 70,A -42.3136,B 24.8916,C -2.4029,E1 25.1284,E2 126.3971} C_DIS
LIN {X 49.1663,Y -39.112,Z 70,A -45.0279,B 24.8927,C -2.3908,E1 25.1237,E2 129.1273} C_DIS
LIN {X 46.961,Y -41.7342,Z 70,A -48.0481,B 24.8932,C -2.3854,E1 25.1182,E2 132.1466} C_DIS
LIN {X 44.4882,Y -44.3612,Z 70,A -50.9189,B 24.893,C -2.3876,E1 25.1127,E2 134.9998} C_DIS
LIN {X 42.1425,Y -46.5938,Z 70,A -54.4091,B 24.8948,C -2.3677,E1 25.1055,E2 138.5227} C_DIS
LIN {X 39.0907,Y -49.1816,Z 70,A -58.1929,B 24.8958,C -2.3566,E1 25.0973,E2 142.3185} C_DIS
LIN {X 35.6369,Y -51.7408,Z 70,A -61.4581,B 24.8951,C -2.3642,E1 25.09,E2 145.5541} C_DIS
LIN {X 33.6941,Y -53.0266,Z 70,A -63.7724,B 24.8959,C -2.3556,E1 25.0845,E2 147.8811} C_DIS
LIN {X 30.9053,Y -54.6991,Z 70,A -66.8558,B 24.8966,C -2.3475,E1 25.077,E2 150.9744} C_DIS
LIN {X 28.8945,Y -55.7876,Z 70,A -68.923,B 24.8969,C -2.3445,E1 25.0719,E2 153.0431} C_DIS
LIN {X 26.2599,Y -57.0747,Z 70,A -71.4907,B 24.897,C -2.3428,E1 25.0655,E2 155.6081} C_DIS
LIN {X 22.9713,Y -58.4752,Z 70,A -74.769,B 24.8975,C -2.3378,E1 25.057,E2 158.8907} C_DIS
LIN {X 20.2578,Y -59.4701,Z 70,A -77.3846,B 24.8977,C -2.3349,E1 25.0501,E2 161.5079} C_DIS
LIN {X 17.4819,Y -60.3452,Z 70,A -80.7153,B 24.8993,C -2.3164,E1 25.0411,E2 164.8765} C_DIS
LIN {X 14.0427,Y -61.236,Z 70,A -83.218,B 24.8981,C -2.3301,E1 25.0344,E2 167.3432} C_DIS
LIN {X 10.5885,Y -61.9271,Z 70,A -86.4128,B 24.8983,C -2.3279,E1 25.0256,E2 170.5397} C_DIS
LIN {X 7.8752,Y -62.3302,Z 70,A -88.9598,B 24.8986,C -2.3252,E1 25.0186,E2 173.0909} C_DIS
LIN {X 5.0379,Y -62.6231,Z 70,A -91.577,B 24.8987,C -2.3235,E1 25.0113,E2 175.7105} C_DIS
LIN {X 1.8918,Y -62.7969,Z 70,A -94.311,B 24.8985,C -2.3255,E1 25.0037,E2 178.4388} C_DIS
LIN {X 1.8918,Y -62.7969,Z 70,A -94.311,B 24.8985,C -2.3255,E1 25.0037,E2 178.4388} C_DIS
Enddeposition()
LIN {X 0.4029,Y -61.8721,Z 70,A -95.8124,B 24.8974,C -2.3387,E1 24.9996,E2 179.9087} C_DIS
Startdeposition()
$VEL.CP = VEL_PRINT
LIN {X 2.5989,Y -61.8194,Z 70,A -92.1118,B 24.894,C -2.3762,E1 25.0101,E2 176.1198} C_DIS
LIN {X 6.4733,Y -61.5344,Z 70,A -88.8967,B 24.8947,C -2.3694,E1 25.019,E2 172.9227} C_DIS
LIN {X 9.3945,Y -61.1566,Z 70,A -86.7414,B 24.8956,C -2.3583,E1 25.0249,E2 170.7957} C_DIS
LIN {X 13.8128,Y -60.3126,Z 70,A -82.2695,B 24.8947,C -2.3687,E1 25.0372,E2 166.3045} C_DIS
LIN {X 16.3831,Y -59.666,Z 70,A -79.3193,B 24.8935,C -2.3826,E1 25.0453,E2 163.3258} C_DIS
LIN {X 20.9779,Y -58.2097,Z 70,A -74.7706,B 24.8928,C -2.3901,E1 25.0573,E2 158.7683} C_DIS
LIN {X 24.8885,Y -56.6479,Z 70,A -71.1828,B 24.893,C -2.3883,E1 25.0665,E2 155.1931} C_DIS
LIN {X 27.6322,Y -55.3614,Z 70,A -68.4245,B 24.8927,C -2.3916,E1 25.0734,E2 152.4342} C_DIS
LIN {X 30.3723,Y -53.907,Z 70,A -65.4574,B 24.892,C -2.3988,E1 25.0807,E2 149.4587} C_DIS
LIN {X 33.0485,Y -52.3095,Z 70,A -62.7479,B 24.892,C -2.3999,E1 25.0872,E2 146.7551} C_DIS
LIN {X 35.6375,Y -50.5814,Z 70,A -59.7708,B 24.8912,C -2.4079,E1 25.094,E2 143.7693} C_DIS
LIN {X 38.6231,Y -48.3377,Z 70,A -56.4112,B 24.8907,C -2.4128,E1 25.1015,E2 140.4103} C_DIS
LIN {X 41.2544,Y -46.1136,Z 70,A -52.9629,B 24.8895,C -2.4263,E1 25.1088,E2 136.9438} C_DIS
LIN {X 43.5545,Y -43.9477,Z 70,A -50.5557,B 24.89,C -2.4205,E1 25.1135,E2 134.5602} C_DIS
LIN {X 45.4191,Y -42.0185,Z 70,A -47.8631,B 24.889,C -2.4317,E1 25.1187,E2 131.8529} C_DIS
LIN {X 47.2812,Y -39.9116,Z 70,A -45.0864,B 24.888,C -2.4426,E1 25.1238,E2 129.0631} C_DIS
LIN {X 49.3629,Y -37.3058,Z 70,A -42.271,B 24.888,C -2.444,E1 25.1286,E2 126.2577} C_DIS
LIN {X 51.3658,Y -34.4964,Z 70,A -38.9966,B 24.8869,C -2.4546,E1 25.1339,E2 122.9741} C_DIS
LIN {X 53.0184,Y -31.8985,Z 70,A -36.1591,B 24.8862,C -2.4623,E1 25.138,E2 120.1329} C_DIS
LIN {X 54.4213,Y -29.4399,Z 70,A -33.2966,B 24.8849,C -2.4758,E1 25.1419,E2 117.2532} C_DIS
LIN {X 55.9056,Y -26.5144,Z 70,A -30.7224,B 24.8852,C -2.4732,E1 25.1451,E2 114.6992} C_DIS
LIN {X 57.0914,Y -23.8525,Z 70,A -27.4253,B 24.883,C -2.4962,E1 25.1487,E2 111.3656} C_DIS
LIN {X 58.8506,Y -19.1051,Z 70,A -22.6958,B 24.8816,C -2.5116,E1 25.1531,E2 106.6265} C_DIS
LIN {X 59.932,Y -15.3799,Z 70,A -18.6434,B 24.8794,C -2.5344,E1 25.1559,E2 102.5433} C_DIS
LIN {X 60.7614,Y -11.6809,Z 70,A -16.1682,B 24.8809,C -2.5192,E1 25.1573,E2 100.1185} C_DIS
LIN {X 61.2437,Y -8.8097,Z 70,A -13.8496,B 24.8809,C -2.5183,E1 25.1583,E2 97.8158} C_DIS
LIN {X 61.6211,Y -5.5891,Z 70,A -10.3699,B 24.8789,C -2.5398,E1 25.1593,E2 94.306} C_DIS
LIN {X 61.834,Y -2.2515,Z 70,A -7.4374,B 24.8784,C -2.5454,E1 25.1597,E2 91.3775} C_DIS
LIN {X 61.871,Y 0.7019,Z 70,A -4.6968,B 24.8775,C -2.5542,E1 25.1597,E2 88.6324} C_DIS
LIN {X 61.6823,Y 4.8667,Z 70,A -1.1605,B 24.8771,C -2.5582,E1 25.1592,E2 85.1077} C_DIS
LIN {X 61.1006,Y 9.7567,Z 70,A 3.649,B 24.8752,C -2.5785,E1 25.1575,E2 80.2785} C_DIS
LIN {X 59.9661,Y 15.2474,Z 70,A 8.7957,B 24.8737,C -2.5932,E1 25.1544,E2 75.1271} C_DIS
LIN {X 58.7224,Y 19.4975,Z 70,A 12.5147,B 24.8735,C -2.5958,E1 25.1514,E2 71.423} C_DIS
LIN {X 57.7196,Y 22.2927,Z 70,A 15.9497,B 24.871,C -2.6207,E1 25.148,E2 67.9483} C_DIS
LIN {X 56.247,Y 25.7835,Z 70,A 19.0179,B 24.8711,C -2.6197,E1 25.1446,E2 64.8993} C_DIS
LIN {X 54.9734,Y 28.397,Z 70,A 22.3281,B 24.8689,C -2.6423,E1 25.1404,E2 61.5533} C_DIS
LIN {X 52.3393,Y 33.0007,Z 70,A 26.3287,B 24.8699,C -2.6328,E1 25.1347,E2 57.5957} C_DIS
LIN {X 50.3632,Y 35.9435,Z 70,A 29.8891,B 24.8684,C -2.6477,E1 25.1291,E2 54.0176} C_DIS
LIN {X 48.6568,Y 38.2222,Z 70,A 32.5134,B 24.8678,C -2.6536,E1 25.1246,E2 51.3916} C_DIS
LIN {X 46.8588,Y 40.4076,Z 70,A 35.6942,B 24.8658,C -2.6731,E1 25.1188,E2 48.1792} C_DIS
LIN {X 43.0409,Y 44.451,Z 70,A 41.0363,B 24.8643,C -2.6886,E1 25.1083,E2 42.8232} C_DIS
LIN {X 40.6838,Y 46.6178,Z 70,A 43.2076,B 24.8656,C -2.6754,E1 25.1038,E2 40.6917} C_DIS
LIN {X 38.4831,Y 48.4506,Z 70,A 45.7145,B 24.8654,C -2.6769,E1 25.0984,E2 38.1909} C_DIS
LIN {X 36.3121,Y 50.098,Z 70,A 48.1965,B 24.8651,C -2.6802,E1 25.0929,E2 35.7097} C_DIS
LIN {X 34.6146,Y 51.2857,Z 70,A 50.2705,B 24.8644,C -2.687,E1 25.0881,E2 33.6268} C_DIS
LIN {X 32.0993,Y 52.8964,Z 70,A 52.9608,B 24.8642,C -2.6894,E1 25.0817,E2 30.9394} C_DIS
LIN {X 28.271,Y 55.0377,Z 70,A 57.0698,B 24.8635,C -2.6959,E1 25.0716,E2 26.8269} C_DIS
LIN {X 26.5521,Y 55.8878,Z 70,A 58.958,B 24.863,C -2.7005,E1 25.0668,E2 24.9326} C_DIS
LIN {X 24.4736,Y 56.8287,Z 70,A 61.0725,B 24.8628,C -2.7029,E1 25.0614,E2 22.8176} C_DIS
LIN {X 21.6745,Y 57.954,Z 70,A 63.8034,B 24.8627,C -2.7041,E1 25.0543,E2 20.0898} C_DIS
LIN {X 18.5624,Y 59.0244,Z 70,A 66.7541,B 24.8627,C -2.7044,E1 25.0465,E2 17.1441} C_DIS
LIN {X 15.4087,Y 59.9246,Z 70,A 69.9266,B 24.8621,C -2.7093,E1 25.0379,E2 13.9649} C_DIS
LIN {X 11.8362,Y 60.7306,Z 70,A 73.7742,B 24.8609,C -2.721,E1 25.0274,E2 10.0944} C_DIS
LIN {X 8.2819,Y 61.3175,Z 70,A 77.525,B 24.8599,C -2.731,E1 25.0169,E2 6.3231} C_DIS
LIN {X 4.6371,Y 61.7007,Z 70,A 79.9352,B 24.8621,C -2.7097,E1 25.0104,E2 3.9649} C_DIS
LIN {X 0.3187,Y 61.8732,Z 70,A 83.9698,B 24.8621,C -2.7099,E1 24.9991,E2 -0.0696} C_DIS
LIN {X -2.5611,Y 61.821,Z 70,A 86.3361,B 24.8628,C -2.7028,E1 24.9925,E2 -2.4192} C_DIS
LIN {X -6.1147,Y 61.5712,Z 70,A 89.584,B 24.8631,C -2.7003,E1 24.9835,E2 -5.6624} C_DIS
LIN {X -7.639,Y 61.4014,Z 70,A 91.4764,B 24.8621,C -2.7093,E1 24.9782,E2 -7.5777} C_DIS
LIN {X -11.1328,Y 60.8645,Z 70,A 94.462,B 24.863,C -2.701,E1 24.97,E2 -10.5463} C_DIS
LIN {X -14.8183,Y 60.0735,Z 70,A 98.6177,B 24.8619,C -2.7117,E1 24.9586,E2 -14.7328} C_DIS
LIN {X -18.0984,Y 59.1683,Z 70,A 101.6331,B 24.8625,C -2.7055,E1 24.9506,E2 -17.7384} C_DIS
LIN {X -22.5383,Y 57.6231,Z 70,A 105.9181,B 24.8632,C -2.6985,E1 24.9394,E2 -22.0156} C_DIS
LIN {X -27.5919,Y 55.3813,Z 70,A 110.8202,B 24.8645,C -2.6864,E1 24.927,E2 -26.9011} C_DIS
LIN {X -30.2443,Y 53.9785,Z 70,A 113.584,B 24.865,C -2.6815,E1 24.9202,E2 -29.661} C_DIS
LIN {X -32.7164,Y 52.517,Z 70,A 115.9656,B 24.866,C -2.6712,E1 24.9146,E2 -32.0254} C_DIS
LIN {X -35.7766,Y 50.4823,Z 70,A 119.9656,B 24.8655,C -2.6763,E1 24.9053,E2 -36.051} C_DIS
LIN {X -38.6736,Y 48.2997,Z 70,A 123.0406,B 24.8668,C -2.6638,E1 24.8986,E2 -39.1073} C_DIS
LIN {X -41.006,Y 46.336,Z 70,A 125.8797,B 24.8674,C -2.6578,E1 24.8926,E2 -41.9433} C_DIS
LIN {X -42.401,Y 45.0616,Z 70,A 127.9041,B 24.8672,C -2.6591,E1 24.8884,E2 -43.979} C_DIS
LIN {X -45.4177,Y 42.02,Z 70,A 131.5837,B 24.8687,C -2.644,E1 24.8813,E2 -47.6385} C_DIS
LIN {X -47.3902,Y 39.7825,Z 70,A 134.3663,B 24.8694,C -2.6375,E1 24.8763,E2 -50.4181} C_DIS
LIN {X -49.0783,Y 37.6792,Z 70,A 137.3542,B 24.8691,C -2.6403,E1 24.8711,E2 -53.4269} C_DIS
LIN {X -51.1593,Y 34.8013,Z 70,A 140.0669,B 24.8711,C -2.6205,E1 24.8668,E2 -56.1057} C_DIS
LIN {X -53.1403,Y 31.6948,Z 70,A 143.6362,B 24.8717,C -2.614,E1 24.8615,E2 -59.6775} C_DIS
LIN {X -54.5963,Y 29.1159,Z 70,A 146.064,B 24.8731,C -2.6003,E1 24.8583,E2 -62.0853} C_DIS
LIN {X -55.8402,Y 26.6512,Z 70,A 149.4304,B 24.8723,C -2.6079,E1 24.8541,E2 -65.4882} C_DIS
LIN {X -57.3667,Y 23.1834,Z 70,A 153.0416,B 24.8731,C -2.5993,E1 24.8502,E2 -69.0989} C_DIS
LIN {X -58.7934,Y 19.2816,Z 70,A 156.4393,B 24.8751,C -2.5792,E1 24.8472,E2 -72.4679} C_DIS
LIN {X -59.4657,Y 17.0959,Z 70,A 158.7835,B 24.8753,C -2.5769,E1 24.8453,E2 -74.8201} C_DIS
LIN {X -60.2515,Y 14.0771,Z 70,A 161.2765,B 24.8769,C -2.5606,E1 24.8437,E2 -77.2887} C_DIS
LIN {X -60.7479,Y 11.7507,Z 70,A 163.6184,B 24.8773,C -2.5563,E1 24.8424,E2 -79.6341} C_DIS
LIN {X -61.2148,Y 9.0094,Z 70,A 166.2755,B 24.878,C -2.5497,E1 24.8412,E2 -82.2913} C_DIS
LIN {X -61.5704,Y 6.13,Z 70,A 168.9979,B 24.8787,C -2.5418,E1 24.8404,E2 -85.0112} C_DIS
LIN {X -61.8203,Y 2.5773,Z 70,A 172.0515,B 24.8801,C -2.5269,E1 24.8399,E2 -88.0476} C_DIS
LIN {X -61.8752,Y 0.2359,Z 70,A 174.7655,B 24.8798,C -2.5301,E1 24.8398,E2 -90.7855} C_DIS
LIN {X -61.7498,Y -3.9257,Z 70,A 178.0057,B 24.8821,C -2.5066,E1 24.8402,E2 -93.9891} C_DIS
LIN {X -61.3738,Y -7.8517,Z 70,A -177.4711,B 24.8816,C -2.5114,E1 24.8416,E2 -98.5509} C_DIS
LIN {X -60.7002,Y -11.9987,Z 70,A -174.036,B 24.8835,C -2.491,E1 24.8432,E2 -101.9574} C_DIS
LIN {X -60.0674,Y -14.8436,Z 70,A -171.3098,B 24.8842,C -2.4833,E1 24.845,E2 -104.6813} C_DIS
LIN {X -59.3099,Y -17.6275,Z 70,A -168.5499,B 24.8848,C -2.477,E1 24.8471,E2 -107.4422} C_DIS
LIN {X -58.3689,Y -20.5296,Z 70,A -165.8547,B 24.8858,C -2.4664,E1 24.8495,E2 -110.1272} C_DIS
LIN {X -57.4321,Y -23.0227,Z 70,A -163.4362,B 24.8866,C -2.4584,E1 24.8519,E2 -112.5402} C_DIS
LIN {X -55.982,Y -26.3528,Z 70,A -159.9232,B 24.8872,C -2.4518,E1 24.856,E2 -116.0568} C_DIS
LIN {X -54.8807,Y -28.5759,Z 70,A -157.318,B 24.8872,C -2.4515,E1 24.8593,E2 -118.6751} C_DIS
LIN {X -53.0742,Y -31.8058,Z 70,A -154.0116,B 24.8882,C -2.4402,E1 24.8639,E2 -121.9718} C_DIS
LIN {X -51.415,Y -34.4237,Z 70,A -151.2319,B 24.8891,C -2.4312,E1 24.8682,E2 -124.7439} C_DIS
LIN {X -49.6307,Y -36.9493,Z 70,A -148.0956,B 24.8892,C -2.4296,E1 24.8733,E2 -127.8915} C_DIS
LIN {X -47.3379,Y -39.8452,Z 70,A -144.8852,B 24.8903,C -2.4176,E1 24.879,E2 -131.0883} C_DIS
LIN {X -44.98,Y -42.4878,Z 70,A -141.5865,B 24.8909,C -2.4108,E1 24.8852,E2 -134.3854} C_DIS
LIN {X -42.6667,Y -44.8116,Z 70,A -138.5909,B 24.8916,C -2.4038,E1 24.8912,E2 -137.3767} C_DIS
LIN {X -40.5486,Y -46.7358,Z 70,A -136.1291,B 24.8924,C -2.3949,E1 24.8963,E2 -139.8273} C_DIS
LIN {X -38.2062,Y -48.6693,Z 70,A -133.0783,B 24.8924,C -2.3946,E1 24.9029,E2 -142.8887} C_DIS
LIN {X -35.3581,Y -50.776,Z 70,A -129.7327,B 24.8928,C -2.3905,E1 24.9105,E2 -146.2361} C_DIS
LIN {X -32.8856,Y -52.4113,Z 70,A -127.0096,B 24.8932,C -2.3859,E1 24.9169,E2 -148.957} C_DIS
LIN {X -30.1864,Y -54.0109,Z 70,A -124.4207,B 24.8941,C -2.3754,E1 24.9231,E2 -151.5286} C_DIS
LIN {X -27.8309,Y -55.2627,Z 70,A -122.0001,B 24.8945,C -2.3712,E1 24.9291,E2 -153.946} C_DIS
LIN {X -25.8234,Y -56.2274,Z 70,A -119.6826,B 24.8942,C -2.3742,E1 24.935,E2 -156.2763} C_DIS
LIN {X -23.2037,Y -57.3585,Z 70,A -116.8531,B 24.8942,C -2.3754,E1 24.9423,E2 -159.1152} C_DIS
LIN {X -20.2917,Y -58.4524,Z 70,A -113.8001,B 24.894,C -2.3766,E1 24.9504,E2 -162.1771} C_DIS
LIN {X -16.5462,Y -59.6215,Z 70,A -110.6222,B 24.8951,C -2.3644,E1 24.9588,E2 -165.3313} C_DIS
LIN {X -14.5393,Y -60.1416,Z 70,A -108.4596,B 24.8947,C -2.3686,E1 24.9647,E2 -167.5069} C_DIS
LIN {X -11.7501,Y -60.7481,Z 70,A -104.8283,B 24.8929,C -2.3891,E1 24.9748,E2 -171.191} C_DIS
LIN {X -7.9572,Y -61.3602,Z 70,A -102.3415,B 24.8951,C -2.3648,E1 24.9815,E2 -173.6221} C_DIS
LIN {X -3.9949,Y -61.7451,Z 70,A -98.6116,B 24.895,C -2.3656,E1 24.9919,E2 -177.3557} C_DIS
LIN {X -1.0454,Y -61.8652,Z 70,A -95.8772,B 24.895,C -2.366,E1 24.9996,E2 -180.0913} C_DIS
LIN {X -1.0454,Y -61.8652,Z 70,A -95.8772,B 24.895,C -2.366,E1 24.9996,E2 -180.0913} C_DIS
Enddeposition()
LIN {X 0.3741,Y -60.9214,Z 70,A -95.426,B 24.8951,C -2.3639,E1 25.0008,E2 -180.5374} C_DIS
Startdeposition()
$VEL.CP = VEL_PRINT
LIN {X -1.6114,Y -60.9018,Z 70,A -97.7434,B 24.896,C -2.3539,E1 24.9943,E2 -178.1962} C_DIS
LIN {X -6.2648,Y -60.5996,Z 70,A -101.7468,B 24.8953,C -2.362,E1 24.9832,E2 -174.2105} C_DIS
LIN {X -9.8259,Y -60.1254,Z 70,A -105.6439,B 24.8962,C -2.3519,E1 24.9723,E2 -170.2862} C_DIS
LIN {X -12.2108,Y -59.6863,Z 70,A -108.1697,B 24.8966,C -2.3478,E1 24.9654,E2 -167.7477} C_DIS
LIN {X -16.2305,Y -58.7218,Z 70,A -111.8186,B 24.896,C -2.3548,E1 24.9555,E2 -164.1102} C_DIS
LIN {X -19.5348,Y -57.7057,Z 70,A -114.7434,B 24.8951,C -2.3639,E1 24.9478,E2 -161.2018} C_DIS
LIN {X -21.8212,Y -56.8809,Z 70,A -117.253,B 24.8954,C -2.3614,E1 24.9412,E2 -158.6811} C_DIS
LIN {X -24.3513,Y -55.8442,Z 70,A -120.2973,B 24.896,C -2.3546,E1 24.9333,E2 -155.6136} C_DIS
LIN {X -27.0564,Y -54.5848,Z 70,A -123.1068,B 24.8957,C -2.3579,E1 24.9263,E2 -152.8046} C_DIS
LIN {X -30.066,Y -52.9877,Z 70,A -125.9122,B 24.8946,C -2.3699,E1 24.9195,E2 -150.0198} C_DIS
LIN {X -33.255,Y -51.0468,Z 70,A -130.0611,B 24.8952,C -2.3629,E1 24.9096,E2 -145.8408} C_DIS
LIN {X -36.7352,Y -48.6016,Z 70,A -134.0963,B 24.8947,C -2.369,E1 24.9006,E2 -141.8059} C_DIS
LIN {X -40.179,Y -45.7954,Z 70,A -137.6245,B 24.8929,C -2.3891,E1 24.8931,E2 -138.312} C_DIS
LIN {X -42.2865,Y -43.8567,Z 70,A -140.9253,B 24.8934,C -2.3831,E1 24.8864,E2 -134.9833} C_DIS
LIN {X -46.5045,Y -39.3564,Z 70,A -145.807,B 24.8907,C -2.413,E1 24.8773,E2 -130.1513} C_DIS
LIN {X -48.9549,Y -36.2642,Z 70,A -149.5266,B 24.89,C -2.4215,E1 24.8709,E2 -126.4345} C_DIS
LIN {X -50.8352,Y -33.5758,Z 70,A -153.4376,B 24.8906,C -2.414,E1 24.8647,E2 -122.4861} C_DIS
LIN {X -52.8525,Y -30.3015,Z 70,A -156.2128,B 24.8884,C -2.4388,E1 24.8608,E2 -119.7558} C_DIS
LIN {X -54.7377,Y -26.7481,Z 70,A -161.4803,B 24.8899,C -2.4222,E1 24.854,E2 -114.4205} C_DIS
LIN {X -56.2962,Y -23.2897,Z 70,A -163.8752,B 24.887,C -2.4532,E1 24.8515,E2 -112.0864} C_DIS
LIN {X -57.1988,Y -20.973,Z 70,A -166.3724,B 24.8867,C -2.4571,E1 24.849,E2 -109.5845} C_DIS
LIN {X -58.3908,Y -17.3802,Z 70,A -170.0465,B 24.8859,C -2.4655,E1 24.8459,E2 -105.9095} C_DIS
LIN {X -59.0895,Y -14.8358,Z 70,A -172.4669,B 24.8851,C -2.474,E1 24.8442,E2 -103.4953} C_DIS
LIN {X -59.7377,Y -11.9605,Z 70,A -175.2203,B 24.8843,C -2.4828,E1 24.8426,E2 -100.7466} C_DIS
LIN {X -60.4945,Y -7.2104,Z 70,A -180,B 24.8834,C -2.4923,E1 24.8406,E2 -95.9611} C_DIS
LIN {X -60.8088,Y -3.7357,Z 70,A 176.4671,B 24.8829,C -2.4981,E1 24.8399,E2 -92.4208} C_DIS
LIN {X -60.9116,Y 1.1559,Z 70,A 172.2857,B 24.8808,C -2.52,E1 24.8399,E2 -88.2667} C_DIS
LIN {X -60.7674,Y 4.3484,Z 70,A 169.1913,B 24.88,C -2.528,E1 24.8403,E2 -85.1725} C_DIS
LIN {X -60.5214,Y 6.9805,Z 70,A 166.9046,B 24.879,C -2.5393,E1 24.841,E2 -82.8993} C_DIS
LIN {X -60.2262,Y 9.1857,Z 70,A 164.8131,B 24.8783,C -2.5459,E1 24.8418,E2 -80.8111} C_DIS
LIN {X -59.706,Y 12.1148,Z 70,A 161.4605,B 24.8784,C -2.5449,E1 24.8436,E2 -77.4364} C_DIS
LIN {X -58.4084,Y 17.3209,Z 70,A 156.7998,B 24.8763,C -2.5674,E1 24.8469,E2 -72.8022} C_DIS
LIN {X -57.5525,Y 19.9828,Z 70,A 153.0282,B 24.8774,C -2.5554,E1 24.8504,E2 -68.9804} C_DIS
LIN {X -56.2108,Y 23.4933,Z 70,A 151.0042,B 24.8738,C -2.5926,E1 24.8524,E2 -67.0341} C_DIS
LIN {X -55.3118,Y 25.5381,Z 70,A 148.2857,B 24.8743,C -2.5878,E1 24.8555,E2 -64.2892} C_DIS
LIN {X -53.8098,Y 28.5675,Z 70,A 145.0969,B 24.8734,C -2.5969,E1 24.8596,E2 -61.1049} C_DIS
LIN {X -52.3476,Y 31.1648,Z 70,A 141.6785,B 24.8737,C -2.5939,E1 24.8645,E2 -57.6617} C_DIS
LIN {X -50.175,Y 34.5557,Z 70,A 138.3829,B 24.8718,C -2.6129,E1 24.8695,E2 -54.3953} C_DIS
LIN {X -47.9978,Y 37.5216,Z 70,A 135.4429,B 24.87,C -2.6315,E1 24.8744,E2 -51.4855} C_DIS
LIN {X -45.8782,Y 40.0843,Z 70,A 131.8936,B 24.87,C -2.6318,E1 24.8808,E2 -47.9205} C_DIS
LIN {X -43.4196,Y 42.7353,Z 70,A 127.7637,B 24.8704,C -2.6267,E1 24.8889,E2 -43.7608} C_DIS
LIN {X -40.3659,Y 45.632,Z 70,A 124.5425,B 24.8682,C -2.6492,E1 24.8954,E2 -40.5801} C_DIS
LIN {X -38.1893,Y 47.4677,Z 70,A 121.8093,B 24.8677,C -2.6539,E1 24.9013,E2 -37.8479} C_DIS
LIN {X -36.1667,Y 49.0263,Z 70,A 119.6774,B 24.8667,C -2.6639,E1 24.906,E2 -35.7322} C_DIS
LIN {X -33.7678,Y 50.7083,Z 70,A 116.293,B 24.8674,C -2.6575,E1 24.9139,E2 -32.3211} C_DIS
LIN {X -30.6703,Y 52.6405,Z 70,A 112.735,B 24.867,C -2.6612,E1 24.9224,E2 -28.7612} C_DIS
LIN {X -26.9221,Y 54.6514,Z 70,A 109.337,B 24.8652,C -2.6792,E1 24.9308,E2 -25.3967} C_DIS
LIN {X -24.6951,Y 55.6942,Z 70,A 106.1516,B 24.8665,C -2.6659,E1 24.939,E2 -22.1718} C_DIS
LIN {X -19.8572,Y 57.5953,Z 70,A 101.9148,B 24.8646,C -2.6848,E1 24.95,E2 -17.9713} C_DIS
LIN {X -17.4765,Y 58.3623,Z 70,A 99.8574,B 24.8638,C -2.6932,E1 24.9554,E2 -15.9303} C_DIS
LIN {X -15.045,Y 59.0358,Z 70,A 97.1727,B 24.8642,C -2.6894,E1 24.9627,E2 -13.2326} C_DIS
LIN {X -11.6613,Y 59.7962,Z 70,A 94.1958,B 24.8633,C -2.6978,E1 24.9708,E2 -10.2722} C_DIS
LIN {X -7.6336,Y 60.4427,Z 70,A 90.7203,B 24.8623,C -2.7077,E1 24.9803,E2 -6.8172} C_DIS
LIN {X -3.0741,Y 60.8456,Z 70,A 86.1956,B 24.8626,C -2.7052,E1 24.993,E2 -2.2843} C_DIS
LIN {X 1.0867,Y 60.9129,Z 70,A 81.6316,B 24.8638,C -2.6926,E1 25.0058,E2 2.3096} C_DIS
LIN {X 4.1941,Y 60.7781,Z 70,A 78.7535,B 24.8638,C -2.6936,E1 25.0138,E2 5.1841} C_DIS
LIN {X 8.0052,Y 60.3945,Z 70,A 75.4216,B 24.8632,C -2.6987,E1 25.023,E2 8.5017} C_DIS
LIN {X 10.7933,Y 59.9585,Z 70,A 72.6297,B 24.8636,C -2.6949,E1 25.0307,E2 11.2996} C_DIS
LIN {X 14.0194,Y 59.2884,Z 70,A 69.6832,B 24.8634,C -2.6966,E1 25.0387,E2 14.2382} C_DIS
LIN {X 16.4798,Y 58.6514,Z 70,A 67.3762,B 24.8634,C -2.6969,E1 25.0449,E2 16.5408} C_DIS
LIN {X 18.8062,Y 57.9473,Z 70,A 64.9817,B 24.8638,C -2.6928,E1 25.0513,E2 18.9406} C_DIS
LIN {X 21.4276,Y 57.0302,Z 70,A 61.8613,B 24.8652,C -2.6795,E1 25.0595,E2 22.0862} C_DIS
LIN {X 24.2498,Y 55.8884,Z 70,A 59.0929,B 24.8652,C -2.6785,E1 25.0666,E2 24.8504} C_DIS
LIN {X 27.3886,Y 54.4201,Z 70,A 55.8396,B 24.8657,C -2.6746,E1 25.0748,E2 28.1041} C_DIS
LIN {X 30.7771,Y 52.5775,Z 70,A 52.4134,B 24.8657,C -2.6741,E1 25.0831,E2 31.5215} C_DIS
LIN {X 33.9245,Y 50.604,Z 70,A 49.1934,B 24.8657,C -2.6748,E1 25.0906,E2 34.7292} C_DIS
LIN {X 36.8927,Y 48.4832,Z 70,A 46.0419,B 24.8656,C -2.6753,E1 25.0977,E2 37.8684} C_DIS
LIN {X 38.559,Y 47.1681,Z 70,A 43.5976,B 24.867,C -2.6615,E1 25.1031,E2 40.3362} C_DIS
LIN {X 41.4808,Y 44.6196,Z 70,A 40.3434,B 24.8668,C -2.6633,E1 25.1098,E2 43.573} C_DIS
LIN {X 43.2177,Y 42.9397,Z 70,A 37.6473,B 24.8682,C -2.6489,E1 25.1152,E2 46.292} C_DIS
LIN {X 45.746,Y 40.2356,Z 70,A 34.5787,B 24.8681,C -2.6508,E1 25.121,E2 49.3425} C_DIS
LIN {X 47.1065,Y 38.635,Z 70,A 32.4888,B 24.8688,C -2.6436,E1 25.1247,E2 51.4399} C_DIS
LIN {X 48.7211,Y 36.5762,Z 70,A 29.9558,B 24.8695,C -2.6361,E1 25.129,E2 53.9787} C_DIS
LIN {X 50.6443,Y 33.8642,Z 70,A 26.9099,B 24.8701,C -2.6302,E1 25.1339,E2 57.0236} C_DIS
LIN {X 52.1401,Y 31.5112,Z 70,A 23.202,B 24.8733,C -2.598,E1 25.1393,E2 60.7886} C_DIS
LIN {X 54.0125,Y 28.1826,Z 70,A 20.3101,B 24.8726,C -2.6047,E1 25.1431,E2 63.6495} C_DIS
LIN {X 55.3596,Y 25.4355,Z 70,A 17.8556,B 24.8724,C -2.6068,E1 25.146,E2 66.0859} C_DIS
LIN {X 56.7247,Y 22.2233,Z 70,A 14.3381,B 24.8739,C -2.5919,E1 25.1497,E2 69.6192} C_DIS
LIN {X 57.6322,Y 19.7529,Z 70,A 12.2344,B 24.8737,C -2.5935,E1 25.1516,E2 71.7072} C_DIS
LIN {X 58.4833,Y 17.0656,Z 70,A 9.4771,B 24.8747,C -2.5831,E1 25.1539,E2 74.4733} C_DIS
LIN {X 59.3641,Y 13.6917,Z 70,A 5.7978,B 24.8766,C -2.5637,E1 25.1564,E2 78.1775} C_DIS
LIN {X 60.1134,Y 9.8972,Z 70,A 2.2884,B 24.8774,C -2.5556,E1 25.1581,E2 81.6854} C_DIS
LIN {X 60.6804,Y 5.4289,Z 70,A -1.1986,B 24.8769,C -2.5605,E1 25.1592,E2 85.1401} C_DIS
LIN {X 60.9044,Y 1.527,Z 70,A -5.1521,B 24.8787,C -2.5422,E1 25.1598,E2 89.1135} C_DIS
LIN {X 60.9098,Y -1.2532,Z 70,A -7.8631,B 24.8797,C -2.5316,E1 25.1597,E2 91.8334} C_DIS
LIN {X 60.7639,Y -4.3916,Z 70,A -10.6088,B 24.8801,C -2.5273,E1 25.1593,E2 94.5728} C_DIS
LIN {X 60.4946,Y -7.2093,Z 70,A -13.744,B 24.882,C -2.5074,E1 25.1583,E2 97.7365} C_DIS
LIN {X 60.0717,Y -10.1468,Z 70,A -16.8028,B 24.8834,C -2.4922,E1 25.1569,E2 100.8134} C_DIS
LIN {X 58.9307,Y -15.4535,Z 70,A -20.7956,B 24.8824,C -2.5031,E1 25.1545,E2 104.7571} C_DIS
LIN {X 58.0522,Y -18.4808,Z 70,A -24.7417,B 24.8855,C -2.4702,E1 25.1512,E2 108.7585} C_DIS
LIN {X 56.8683,Y -21.8549,Z 70,A -27.6538,B 24.8855,C -2.4708,E1 25.1484,E2 111.6529} C_DIS
LIN {X 55.3664,Y -25.4208,Z 70,A -31.085,B 24.886,C -2.465,E1 25.1446,E2 115.0791} C_DIS
LIN {X 53.4106,Y -29.3079,Z 70,A -35.2734,B 24.8873,C -2.4508,E1 25.1392,E2 119.279} C_DIS
LIN {X 51.8765,Y -31.9455,Z 70,A -38.0902,B 24.8879,C -2.4439,E1 25.1352,E2 122.0975} C_DIS
LIN {X 49.5104,Y -35.5007,Z 70,A -42.3484,B 24.8894,C -2.4272,E1 25.1284,E2 126.3743} C_DIS
LIN {X 47.547,Y -38.0914,Z 70,A -45.6818,B 24.8908,C -2.4126,E1 25.1226,E2 129.7265} C_DIS
LIN {X 45.0074,Y -41.0599,Z 70,A -48.751,B 24.8903,C -2.4177,E1 25.117,E2 132.77} C_DIS
LIN {X 42.8772,Y -43.2795,Z 70,A -51.4206,B 24.8905,C -2.416,E1 25.1118,E2 135.4323} C_DIS
LIN {X 41.6125,Y -44.4961,Z 70,A -53.3819,B 24.8915,C -2.4048,E1 25.1078,E2 137.4119} C_DIS
LIN {X 39.158,Y -46.6722,Z 70,A -56.3731,B 24.8919,C -2.4001,E1 25.1015,E2 140.4026} C_DIS
LIN {X 36.749,Y -48.5912,Z 70,A -59.6142,B 24.8932,C -2.386,E1 25.0943,E2 143.6651} C_DIS
LIN {X 32.7079,Y -51.3985,Z 70,A -63.5269,B 24.8925,C -2.3934,E1 25.0853,E2 147.547} C_DIS
LIN {X 30.9883,Y -52.4527,Z 70,A -65.6891,B 24.8934,C -2.3838,E1 25.0801,E2 149.7252} C_DIS
LIN {X 29.0012,Y -53.5769,Z 70,A -67.6393,B 24.8933,C -2.3846,E1 25.0753,E2 151.6678} C_DIS
LIN {X 26.9153,Y -54.6548,Z 70,A -70.492,B 24.8949,C -2.3664,E1 25.0681,E2 154.5559} C_DIS
LIN {X 22.5607,Y -56.5909,Z 70,A -74.5561,B 24.8947,C -2.3693,E1 25.0577,E2 158.6034} C_DIS
LIN {X 20.2661,Y -57.453,Z 70,A -77.3844,B 24.896,C -2.3547,E1 25.0502,E2 161.4606} C_DIS
LIN {X 14.9184,Y -59.0683,Z 70,A -82.7452,B 24.8967,C -2.3468,E1 25.0358,E2 166.8315} C_DIS
LIN {X 9.1417,Y -60.233,Z 70,A -87.369,B 24.8953,C -2.3624,E1 25.0232,E2 171.4128} C_DIS
LIN {X 4.7261,Y -60.7391,Z 70,A -91.8004,B 24.896,C -2.3546,E1 25.0109,E2 175.8599} C_DIS
LIN {X 0.3741,Y -60.9214,Z 70,A -93.9427,B 24.8923,C -2.3958,E1 25.0052,E2 177.9038} C_DIS
Enddeposition()
LIN {X 0.3741,Y -60.9214,Z 70,A -93.9427,B 24.8923,C -2.3958,E1 25.0052,E2 177.9038} C_DIS
Startdeposition()
$VEL.CP = VEL_PRINT
LIN {X 4.0341,Y -59.8353,Z 70,A -91.7092,B 24.8932,C -2.3857,E1 25.0113,E2 175.6949} C_DIS
LIN {X 6.281,Y -59.6413,Z 70,A -88.7792,B 24.8916,C -2.4037,E1 25.0196,E2 172.724} C_DIS
LIN {X 9.6917,Y -59.1832,Z 70,A -85.2948,B 24.891,C -2.4103,E1 25.0292,E2 169.2271} C_DIS
LIN {X 14.2006,Y -58.2656,Z 70,A -81.5536,B 24.8919,C -2.3997,E1 25.0394,E2 165.516} C_DIS
LIN {X 17.4376,Y -57.3807,Z 70,A -77.7421,B 24.8904,C -2.4168,E1 25.0497,E2 161.6705} C_DIS
LIN {X 20.4697,Y -56.3696,Z 70,A -75.2892,B 24.8913,C -2.4071,E1 25.0561,E2 159.2455} C_DIS
LIN {X 22.8011,Y -55.4679,Z 70,A -72.42,B 24.89,C -2.4213,E1 25.0636,E2 156.3492} C_DIS
LIN {X 27.4134,Y -53.3391,Z 70,A -67.8518,B 24.8899,C -2.4224,E1 25.075,E2 151.7903} C_DIS
LIN {X 30.0513,Y -51.8989,Z 70,A -65.0298,B 24.8895,C -2.4262,E1 25.0819,E2 148.9674} C_DIS
LIN {X 32.5396,Y -50.376,Z 70,A -61.9472,B 24.8884,C -2.4383,E1 25.0892,E2 145.8662} C_DIS
LIN {X 36.5435,Y -47.5512,Z 70,A -57.1043,B 24.8872,C -2.4517,E1 25.1002,E2 141.0087} C_DIS
LIN {X 39.4419,Y -45.176,Z 70,A -54.0627,B 24.8876,C -2.4469,E1 25.1066,E2 137.9903} C_DIS
LIN {X 41.3132,Y -43.4724,Z 70,A -51.6442,B 24.8871,C -2.4525,E1 25.1115,E2 135.5684} C_DIS
LIN {X 43.0572,Y -41.745,Z 70,A -49.3256,B 24.8866,C -2.4576,E1 25.1161,E2 133.2478} C_DIS
LIN {X 44.5991,Y -40.0933,Z 70,A -47.2944,B 24.8864,C -2.4599,E1 25.1199,E2 131.22} C_DIS
LIN {X 46.6332,Y -37.7078,Z 70,A -44.3799,B 24.8859,C -2.4657,E1 25.1252,E2 128.3052} C_DIS
LIN {X 48.8567,Y -34.7787,Z 70,A -40.3827,B 24.8839,C -2.4866,E1 25.1318,E2 124.2776} C_DIS
LIN {X 51.0844,Y -31.4169,Z 70,A -36.7699,B 24.8835,C -2.4915,E1 25.1373,E2 120.6714} C_DIS
LIN {X 52.396,Y -29.1753,Z 70,A -34.0245,B 24.8822,C -2.505,E1 25.1411,E2 117.9084} C_DIS
LIN {X 54.4534,Y -25.1278,Z 70,A -29.8889,B 24.8815,C -2.5128,E1 25.1461,E2 113.7765} C_DIS
LIN {X 55.7583,Y -22.081,Z 70,A -27.0829,B 24.8815,C -2.5136,E1 25.1491,E2 110.9841} C_DIS
LIN {X 56.4373,Y -20.2842,Z 70,A -24.7061,B 24.8796,C -2.5323,E1 25.1514,E2 108.5763} C_DIS
LIN {X 57.8248,Y -15.903,Z 70,A -20.8901,B 24.8796,C -2.5319,E1 25.1545,E2 104.7831} C_DIS
LIN {X 58.5987,Y -12.7565,Z 70,A -17.2376,B 24.8774,C -2.5552,E1 25.1568,E2 101.0967} C_DIS
LIN {X 59.2151,Y -9.4988,Z 70,A -14.1958,B 24.8768,C -2.562,E1 25.1582,E2 98.0566} C_DIS
LIN {X 59.6308,Y -6.3814,Z 70,A -11.6773,B 24.877,C -2.5597,E1 25.159,E2 95.5586} C_DIS
LIN {X 59.8497,Y -3.8207,Z 70,A -8.7757,B 24.8752,C -2.5783,E1 25.1596,E2 92.63} C_DIS
LIN {X 59.973,Y -0.1662,Z 70,A -5.818,B 24.8754,C -2.5763,E1 25.1598,E2 89.6948} C_DIS
LIN {X 59.9096,Y 2.7204,Z 70,A -2.4191,B 24.873,C -2.6006,E1 25.1594,E2 86.2586} C_DIS
LIN {X 59.6331,Y 6.3545,Z 70,A 1.5772,B 24.8707,C -2.6241,E1 25.1583,E2 82.2304} C_DIS
LIN {X 59.1447,Y 9.9218,Z 70,A 3.953,B 24.8722,C -2.6087,E1 25.1573,E2 79.905} C_DIS
LIN {X 58.5778,Y 12.8524,Z 70,A 6.9121,B 24.8711,C -2.62,E1 25.1556,E2 76.9364} C_DIS
LIN {X 57.8343,Y 15.8678,Z 70,A 9.6497,B 24.8708,C -2.6233,E1 25.1537,E2 74.2067} C_DIS
LIN {X 57.2061,Y 18.0017,Z 70,A 12.0301,B 24.8696,C -2.6358,E1 25.1517,E2 71.8105} C_DIS
LIN {X 56.313,Y 20.6249,Z 70,A 15.345,B 24.8672,C -2.6596,E1 25.1485,E2 68.4578} C_DIS
LIN {X 55.1157,Y 23.6415,Z 70,A 17.6595,B 24.8682,C -2.6494,E1 25.1461,E2 66.1801} C_DIS
LIN {X 54.3241,Y 25.4055,Z 70,A 20.1069,B 24.8662,C -2.6689,E1 25.1431,E2 63.6997} C_DIS
LIN {X 51.9361,Y 29.9865,Z 70,A 24.8158,B 24.8655,C -2.6766,E1 25.1368,E2 58.9972} C_DIS
LIN {X 49.2845,Y 34.1699,Z 70,A 28.7933,B 24.8661,C -2.6707,E1 25.1308,E2 55.0535} C_DIS
LIN {X 47.7282,Y 36.3136,Z 70,A 31.6257,B 24.8647,C -2.6839,E1 25.126,E2 52.2036} C_DIS
LIN {X 46.4536,Y 37.9295,Z 70,A 34.1756,B 24.8629,C -2.7022,E1 25.1215,E2 49.6222} C_DIS
LIN {X 44.0179,Y 40.7311,Z 70,A 36.8519,B 24.8641,C -2.6897,E1 25.1166,E2 46.9874} C_DIS
LIN {X 41.5366,Y 43.2581,Z 70,A 39.8723,B 24.8643,C -2.6884,E1 25.1107,E2 43.9828} C_DIS
LIN {X 39.8768,Y 44.7929,Z 70,A 42.374,B 24.863,C -2.7005,E1 25.1055,E2 41.4625} C_DIS
LIN {X 37.5154,Y 46.7892,Z 70,A 45.557,B 24.862,C -2.7112,E1 25.0986,E2 38.2664} C_DIS
LIN {X 33.599,Y 49.6754,Z 70,A 49.9856,B 24.8617,C -2.714,E1 25.0886,E2 33.8466} C_DIS
LIN {X 30.0639,Y 51.8916,Z 70,A 54.6684,B 24.8595,C -2.7355,E1 25.0773,E2 29.1274} C_DIS
LIN {X 26.2826,Y 53.9062,Z 70,A 58.8853,B 24.8586,C -2.7434,E1 25.0668,E2 24.9035} C_DIS
LIN {X 23.0967,Y 55.3455,Z 70,A 61.8509,B 24.8591,C -2.7386,E1 25.0592,E2 21.9563} C_DIS
LIN {X 20.0826,Y 56.5091,Z 70,A 64.5005,B 24.8598,C -2.7318,E1 25.0523,E2 19.3283} C_DIS
LIN {X 17.4233,Y 57.3852,Z 70,A 67.4963,B 24.8589,C -2.7408,E1 25.0443,E2 16.3166} C_DIS
LIN {X 14.2577,Y 58.2517,Z 70,A 70.6825,B 24.8586,C -2.7438,E1 25.0357,E2 13.1283} C_DIS
LIN {X 10.9185,Y 58.9696,Z 70,A 73.7014,B 24.859,C -2.7399,E1 25.0274,E2 10.1222} C_DIS
LIN {X 8.3351,Y 59.3892,Z 70,A 76.0871,B 24.8592,C -2.7382,E1 25.0209,E2 7.7428} C_DIS
LIN {X 5.5634,Y 59.7125,Z 70,A 79.0165,B 24.8586,C -2.7441,E1 25.0127,E2 4.8012} C_DIS
LIN {X 2.9777,Y 59.8981,Z 70,A 81.8836,B 24.8577,C -2.7522,E1 25.0047,E2 1.9159} C_DIS
LIN {X -2.2288,Y 59.9305,Z 70,A 86.0736,B 24.8595,C -2.7348,E1 24.9931,E2 -2.2328} C_DIS
LIN {X -5.2844,Y 59.7381,Z 70,A 89.4531,B 24.8587,C -2.7429,E1 24.9836,E2 -5.6328} C_DIS
LIN {X -8.4257,Y 59.3763,Z 70,A 92.2698,B 24.8593,C -2.7369,E1 24.9758,E2 -8.4374} C_DIS
LIN {X -10.6625,Y 59.0157,Z 70,A 94.1525,B 24.8601,C -2.7297,E1 24.9707,E2 -10.3048} C_DIS
LIN {X -13.0931,Y 58.5253,Z 70,A 96.9812,B 24.8593,C -2.7369,E1 24.9629,E2 -13.1539} C_DIS
LIN {X -15.9306,Y 57.8173,Z 70,A 99.6201,B 24.8599,C -2.731,E1 24.9558,E2 -15.7828} C_DIS
LIN {X -18.5244,Y 57.0385,Z 70,A 102.1226,B 24.8604,C -2.7264,E1 24.9492,E2 -18.2788} C_DIS
LIN {X -21.2013,Y 56.0985,Z 70,A 106.1032,B 24.8582,C -2.748,E1 24.9386,E2 -22.3191} C_DIS
LIN {X -24.9208,Y 54.5489,Z 70,A 108.8108,B 24.8611,C -2.72,E1 24.9319,E2 -24.9664} C_DIS
LIN {X -27.9368,Y 53.0666,Z 70,A 112.2073,B 24.8612,C -2.7184,E1 24.9234,E2 -28.3684} C_DIS
LIN {X -30.8912,Y 51.4039,Z 70,A 114.966,B 24.8627,C -2.7036,E1 24.9168,E2 -31.0999} C_DIS
LIN {X -33.5526,Y 49.7067,Z 70,A 118.5122,B 24.8623,C -2.708,E1 24.9084,E2 -34.668} C_DIS
LIN {X -35.5742,Y 48.2809,Z 70,A 121.6275,B 24.8613,C -2.7174,E1 24.9014,E2 -37.817} C_DIS
LIN {X -38.3439,Y 46.1116,Z 70,A 124.0764,B 24.8638,C -2.693,E1 24.8962,E2 -40.2168} C_DIS
LIN {X -39.9453,Y 44.7316,Z 70,A 126.4382,B 24.8636,C -2.6948,E1 24.8912,E2 -42.5925} C_DIS
LIN {X -42.9559,Y 41.8501,Z 70,A 129.9583,B 24.8654,C -2.6769,E1 24.8843,E2 -46.0845} C_DIS
LIN {X -46.0525,Y 38.415,Z 70,A 134.4784,B 24.8664,C -2.6677,E1 24.876,E2 -50.603} C_DIS
LIN {X -49.2473,Y 34.2234,Z 70,A 139.3327,B 24.868,C -2.6511,E1 24.8679,E2 -55.4409} C_DIS
LIN {X -50.8007,Y 31.8722,Z 70,A 142.49,B 24.868,C -2.6521,E1 24.8631,E2 -58.6165} C_DIS
LIN {X -52.1408,Y 29.6303,Z 70,A 144.4991,B 24.8695,C -2.6363,E1 24.8603,E2 -60.5982} C_DIS
LIN {X -53.4228,Y 27.2496,Z 70,A 147.695,B 24.8692,C -2.6398,E1 24.8561,E2 -63.8196} C_DIS
LIN {X -54.9671,Y 23.9825,Z 70,A 151.3979,B 24.8697,C -2.6341,E1 24.8519,E2 -67.5292} C_DIS
LIN {X -56.8439,Y 19.1131,Z 70,A 155.9011,B 24.8721,C -2.6103,E1 24.8476,E2 -72.001} C_DIS
LIN {X -57.915,Y 15.5689,Z 70,A 159.4812,B 24.8731,C -2.6002,E1 24.8448,E2 -75.5776} C_DIS
LIN {X -58.4204,Y 13.5499,Z 70,A 161.7054,B 24.8733,C -2.5982,E1 24.8434,E2 -77.81} C_DIS
LIN {X -59.129,Y 10.0156,Z 70,A 164.9158,B 24.8747,C -2.5832,E1 24.8417,E2 -81.0036} C_DIS
LIN {X -59.5446,Y 7.1382,Z 70,A 167.7035,B 24.8756,C -2.5747,E1 24.8407,E2 -83.7875} C_DIS
LIN {X -59.867,Y 3.5398,Z 70,A 171.2042,B 24.8765,C -2.5646,E1 24.84,E2 -87.2852} C_DIS
LIN {X -59.9589,Y 1.2173,Z 70,A 173.1116,B 24.8777,C -2.5521,E1 24.8398,E2 -89.1742} C_DIS
LIN {X -59.95,Y -1.6075,Z 70,A 176.4092,B 24.8775,C -2.5542,E1 24.8399,E2 -92.4967} C_DIS
LIN {X -59.7912,Y -4.6399,Z 70,A 179.2244,B 24.8785,C -2.5436,E1 24.8405,E2 -95.3034} C_DIS
LIN {X -59.3666,Y -8.4941,Z 70,A -176.7081,B 24.879,C -2.5386,E1 24.8419,E2 -99.3833} C_DIS
LIN {X -58.6988,Y -12.2901,Z 70,A -173.472,B 24.8809,C -2.5193,E1 24.8436,E2 -102.5924} C_DIS
LIN {X -58.0678,Y -14.9891,Z 70,A -170.4316,B 24.8809,C -2.5184,E1 24.8457,E2 -105.6485} C_DIS
LIN {X -56.5533,Y -19.9568,Z 70,A -165.7769,B 24.8828,C -2.4983,E1 24.8496,E2 -110.2817} C_DIS
LIN {X -55.5669,Y -22.5578,Z 70,A -162.4693,B 24.8824,C -2.5026,E1 24.8531,E2 -113.6181} C_DIS
LIN {X -53.8092,Y -26.479,Z 70,A -158.2623,B 24.8833,C -2.4931,E1 24.8582,E2 -117.8253} C_DIS
LIN {X -52.1705,Y -29.5786,Z 70,A -155.4146,B 24.885,C -2.4749,E1 24.862,E2 -120.6445} C_DIS
LIN {X -49.5082,Y -33.8459,Z 70,A -150.7561,B 24.8864,C -2.46,E1 24.869,E2 -125.2909} C_DIS
LIN {X -48.2781,Y -35.578,Z 70,A -148.2133,B 24.886,C -2.4647,E1 24.8733,E2 -127.8572} C_DIS
LIN {X -45.8545,Y -38.6523,Z 70,A -144.0973,B 24.8861,C -2.4633,E1 24.8807,E2 -131.9889} C_DIS
LIN {X -43.6279,Y -41.1479,Z 70,A -140.9051,B 24.8868,C -2.4564,E1 24.8868,E2 -135.1784} C_DIS
LIN {X -41.2652,Y -43.5176,Z 70,A -138.574,B 24.8889,C -2.4333,E1 24.8914,E2 -137.4641} C_DIS
LIN {X -39.188,Y -45.3978,Z 70,A -136.0033,B 24.8895,C -2.4261,E1 24.8967,E2 -140.0278} C_DIS
LIN {X -36.0091,Y -47.9571,Z 70,A -132.2742,B 24.8905,C -2.4158,E1 24.9049,E2 -143.7463} C_DIS
LIN {X -32.5579,Y -50.3643,Z 70,A -127.1209,B 24.889,C -2.4317,E1 24.9169,E2 -148.9547} C_DIS
LIN {X -29.1,Y -52.4381,Z 70,A -123.2724,B 24.8895,C -2.4264,E1 24.9263,E2 -152.8017} C_DIS
LIN {X -25.9222,Y -54.0794,Z 70,A -120.3759,B 24.8908,C -2.4119,E1 24.9335,E2 -155.6711} C_DIS
LIN {X -22.0748,Y -55.7603,Z 70,A -116.3887,B 24.8912,C -2.4073,E1 24.9437,E2 -159.6567} C_DIS
LIN {X -18.7751,Y -56.9562,Z 70,A -113.1998,B 24.8918,C -2.4012,E1 24.9521,E2 -162.8371} C_DIS
LIN {X -15.9147,Y -57.8216,Z 70,A -110.2275,B 24.8918,C -2.4018,E1 24.9601,E2 -165.8156} C_DIS
LIN {X -12.4453,Y -58.6664,Z 70,A -107.1714,B 24.8926,C -2.3927,E1 24.9684,E2 -168.8541} C_DIS
LIN {X -10.6276,Y -59.0219,Z 70,A -104.9182,B 24.8917,C -2.4022,E1 24.9746,E2 -171.1323} C_DIS
LIN {X -6.1338,Y -59.6567,Z 70,A -100.5354,B 24.8917,C -2.4025,E1 24.9868,E2 -175.5188} C_DIS
LIN {X -1.4494,Y -59.9546,Z 70,A -96.354,B 24.8922,C -2.3964,E1 24.9984,E2 -179.6866} C_DIS
LIN {X 0.3413,Y -59.9615,Z 70,A -93.7678,B 24.8905,C -2.4159,E1 25.0058,E2 -182.319} C_DIS
Enddeposition()
LIN {X 0.3413,Y -59.9615,Z 70,A -93.7678,B 24.8905,C -2.4159,E1 25.0058,E2 -182.319} C_DIS
Startdeposition()
$VEL.CP = VEL_PRINT
LIN {X -0.1733,Y -59.0197,Z 70,A -96.3775,B 24.8931,C -2.3871,E1 24.9983,E2 -179.6411} C_DIS
LIN {X -3.651,Y -58.9076,Z 70,A -100.3046,B 24.8941,C -2.3756,E1 24.9873,E2 -175.6857} C_DIS
LIN {X -6.9824,Y -58.6053,Z 70,A -103.1699,B 24.8934,C -2.3837,E1 24.9794,E2 -172.8379} C_DIS
LIN {X -9.7956,Y -58.2012,Z 70,A -105.9182,B 24.8933,C -2.3846,E1 24.9718,E2 -170.0894} C_DIS
LIN {X -12.6809,Y -57.6414,Z 70,A -108.7795,B 24.8932,C -2.3857,E1 24.964,E2 -167.2272} C_DIS
LIN {X -15.5988,Y -56.9214,Z 70,A -111.5978,B 24.8929,C -2.3893,E1 24.9563,E2 -164.4134} C_DIS
LIN {X -18.0123,Y -56.2037,Z 70,A -113.9121,B 24.8925,C -2.3936,E1 24.9502,E2 -162.1053} C_DIS
LIN {X -19.9017,Y -55.564,Z 70,A -116.0214,B 24.8926,C -2.3918,E1 24.9446,E2 -159.9877} C_DIS
LIN {X -22.3302,Y -54.6324,Z 70,A -118.6823,B 24.8926,C -2.3916,E1 24.9377,E2 -157.3205} C_DIS
LIN {X -25.5031,Y -53.2252,Z 70,A -122.7508,B 24.8935,C -2.3821,E1 24.9273,E2 -153.2192} C_DIS
LIN {X -28.9111,Y -51.4538,Z 70,A -126.6529,B 24.8934,C -2.3838,E1 24.9178,E2 -149.31} C_DIS
LIN {X -31.8604,Y -49.6814,Z 70,A -129.7956,B 24.8926,C -2.3925,E1 24.9104,E2 -146.1779} C_DIS
LIN {X -34.8942,Y -47.5996,Z 70,A -132.8077,B 24.8911,C -2.4088,E1 24.9036,E2 -143.194} C_DIS
LIN {X -37.9921,Y -45.1669,Z 70,A -136.5235,B 24.8903,C -2.4176,E1 24.8956,E2 -139.4855} C_DIS
LIN {X -40.4038,Y -43.0216,Z 70,A -139.2806,B 24.8891,C -2.4307,E1 24.8899,E2 -136.7485} C_DIS
LIN {X -42.9383,Y -40.4924,Z 70,A -143.83,B 24.8902,C -2.4186,E1 24.8809,E2 -132.1507} C_DIS
LIN {X -45.3995,Y -37.7122,Z 70,A -147.1981,B 24.8891,C -2.431,E1 24.8749,E2 -128.7967} C_DIS
LIN {X -47.6014,Y -34.8918,Z 70,A -149.9457,B 24.8871,C -2.4522,E1 24.8703,E2 -126.0865} C_DIS
LIN {X -49.3583,Y -32.359,Z 70,A -153.4436,B 24.8873,C -2.4506,E1 24.8648,E2 -122.5676} C_DIS
LIN {X -50.8429,Y -29.9721,Z 70,A -156.1037,B 24.8865,C -2.4589,E1 24.861,E2 -119.9136} C_DIS
LIN {X -52.847,Y -26.2778,Z 70,A -159.9048,B 24.885,C -2.4747,E1 24.856,E2 -116.1301} C_DIS
LIN {X -54.1873,Y -23.3894,Z 70,A -163.3261,B 24.8848,C -2.4776,E1 24.8521,E2 -112.6969} C_DIS
LIN {X -55.321,Y -20.5679,Z 70,A -166.6311,B 24.8846,C -2.48,E1 24.8488,E2 -109.3791} C_DIS
LIN {X -56.5528,Y -16.8856,Z 70,A -169.9189,B 24.8827,C -2.4994,E1 24.846,E2 -106.1186} C_DIS
LIN {X -57.3223,Y -14.0529,Z 70,A -172.8893,B 24.8821,C -2.5058,E1 24.8439,E2 -103.1464} C_DIS
LIN {X -57.9572,Y -11.1484,Z 70,A -176.0375,B 24.8817,C -2.5102,E1 24.8422,E2 -99.9899} C_DIS
LIN {X -58.553,Y -7.4092,Z 70,A -179.2158,B 24.8798,C -2.53,E1 24.8409,E2 -96.84} C_DIS
LIN {X -58.7636,Y -5.4922,Z 70,A 178.3151,B 24.8803,C -2.5257,E1 24.8402,E2 -94.3459} C_DIS
LIN {X -58.9914,Y -1.828,Z 70,A 175.0831,B 24.8787,C -2.5425,E1 24.8398,E2 -91.1346} C_DIS
LIN {X -59.0121,Y 0.9568,Z 70,A 172.3692,B 24.8778,C -2.5508,E1 24.8398,E2 -88.4244} C_DIS
LIN {X -58.8441,Y 4.5489,Z 70,A 169.0224,B 24.8766,C -2.5643,E1 24.8404,E2 -85.0896} C_DIS
LIN {X -58.6946,Y 6.186,Z 70,A 166.9609,B 24.8768,C -2.5615,E1 24.841,E2 -83.0089} C_DIS
LIN {X -58.1964,Y 9.824,Z 70,A 163.6427,B 24.8753,C -2.5769,E1 24.8423,E2 -79.7077} C_DIS
LIN {X -57.6393,Y 12.6906,Z 70,A 160.8079,B 24.8745,C -2.5857,E1 24.8439,E2 -76.8775} C_DIS
LIN {X -56.5408,Y 16.9246,Z 70,A 156.4971,B 24.8733,C -2.5978,E1 24.8471,E2 -72.5705} C_DIS
LIN {X -55.4694,Y 20.1612,Z 70,A 153.0984,B 24.8725,C -2.6064,E1 24.8502,E2 -69.1729} C_DIS
LIN {X -54.1193,Y 23.5463,Z 70,A 150.0284,B 24.8706,C -2.6249,E1 24.8534,E2 -66.1302} C_DIS
LIN {X -52.8212,Y 26.33,Z 70,A 146.2171,B 24.8712,C -2.6195,E1 24.858,E2 -62.2852} C_DIS
LIN {X -51.18,Y 29.3927,Z 70,A 143.2326,B 24.8696,C -2.6358,E1 24.862,E2 -59.3239} C_DIS
LIN {X -49.7577,Y 31.7416,Z 70,A 140.5885,B 24.8688,C -2.6435,E1 24.8659,E2 -56.6849} C_DIS
LIN {X -47.8,Y 34.6187,Z 70,A 136.6087,B 24.8689,C -2.6423,E1 24.8724,E2 -52.6825} C_DIS
LIN {X -45.7046,Y 37.3426,Z 70,A 133.5786,B 24.8675,C -2.6562,E1 24.8776,E2 -49.6715} C_DIS
LIN {X -43.45,Y 39.9425,Z 70,A 130.4378,B 24.8663,C -2.668,E1 24.8834,E2 -46.5448} C_DIS
LIN {X -40.8897,Y 42.5602,Z 70,A 126.5032,B 24.8662,C -2.6697,E1 24.8912,E2 -42.5977} C_DIS
LIN {X -38.7706,Y 44.4991,Z 70,A 123.316,B 24.8662,C -2.6689,E1 24.898,E2 -39.396} C_DIS
LIN {X -34.6378,Y 47.7873,Z 70,A 118.7457,B 24.8642,C -2.6894,E1 24.908,E2 -34.858} C_DIS
Enddeposition()
END
